(*===================================================================================================*)
(* Monitor reset conditions                                                                          *)
(*===================================================================================================*)
METHOD OkToReset : BOOL
VAR_INPUT
END_VAR
(*===================================================================================================*)
(* Monitor reset conditions                                                                          *)
(*===================================================================================================*)

OkToReset := ((StateAct = NLG_STATUS_STANDBY) AND   // Check for standby mode
			  (ResetCnt < 3));                      // Check reset count is less than 3
END_METHOD

END_FUNCTION_BLOCK

// Application/UserCode/MCU/MCU_Rx
PROGRAM MCU_Rx
VAR
	MCU_CommandResponse1_Rx		:	Receive_CAN1_STD;
	MCU_CommandResponse2_Rx		:	Receive_CAN1_STD;
	MCU_EventInfo1_Rx			:	Receive_CAN1_STD;
	MCU_Info1_Rx				:	Receive_CAN1_STD;
	MCU_Info2_Rx				:	Receive_CAN1_STD;
	MCU_OnEventInfo1_Rx			:	Receive_CAN1_STD;
	MCU_Thermal1_Rx				:	Receive_CAN1_STD;
	MCU_PollingMCUResponse_Rx	:	Receive_CAN1_STD;
	MCU_PollingVMU_Rx			:	Receive_CAN1_STD;
	
	MCU_CommandResponse1_Rx_Timer	:	TON;
	MCU_CommandResponse2_Rx_Timer	:	TON;
	MCU_EventInfo1_Rx_Timer			:	TON;
	MCU_Info1_Rx_Timer				:	TON;
	MCU_Info2_Rx_Timer				:	TON;
	MCU_Thermal1_Rx_Timer			:	TON;
END_VAR


MCU_CommandResponse1_Rx(u32_COBID	:=	16#043,
						 q_NewData => ,
						 au8_Data => ,
						 u8_Length => 			);
						 
MCU_CommandResponse2_Rx(u32_COBID	:=	16#044,
						 q_NewData => ,
						 au8_Data => ,
						 u8_Length => 			);
						 
MCU_EventInfo1_Rx(u32_COBID	:=	16#442,
						 q_NewData => ,
						 au8_Data => ,
						 u8_Length => 			);
						 
MCU_Info1_Rx(u32_COBID	:=	16#440,
						 q_NewData => ,
						 au8_Data => ,
						 u8_Length => 			);
						 
MCU_Info2_Rx(u32_COBID	:=	16#441,
						 q_NewData => ,
						 au8_Data => ,
						 u8_Length => 			);
						 
MCU_OnEventInfo1_Rx(u32_COBID	:=	16#443,
						 q_NewData => ,
						 au8_Data => ,
						 u8_Length => 			);
						 
MCU_Thermal1_Rx(u32_COBID	:=	16#449,
						 q_NewData => ,
						 au8_Data => ,
						 u8_Length => 			);
						 
MCU_PollingMCUResponse_Rx(u32_COBID	:=	16#448,
						 q_NewData => ,
						 au8_Data => ,
						 u8_Length => 			);
						 
MCU_PollingVMU_Rx(u32_COBID	:=	16#445,
						 q_NewData => ,
						 au8_Data => ,
						 u8_Length => 			);
						 


(*MCUCommandResponse1*)
gu8_MCU_State								:=	MCU_CommandResponse1_Rx.au8_Data[0] AND 2#00001111;
gu8_MCU_OperationalMode						:=	MCU_CommandResponse1_Rx.au8_Data[0] AND 2#01110000;
gq_MCU_RegenDeratingStatus					:=	MCU_CommandResponse1_Rx.au8_Data[0].7;
gu8_MCU_RegenDerating						:=	MCU_CommandResponse1_Rx.au8_Data[1] AND 2#00001111;
gu8_MCU_TractionDerating					:=	MCU_CommandResponse1_Rx.au8_Data[1] AND 2#11110000;
gu16_MCU_MaxMotorSpeedForward_Rx			:=	USINT_TO_UINT(MCU_CommandResponse1_Rx.au8_Data[2]) +
												SHL(BOOL_TO_UINT(MCU_CommandResponse1_Rx.au8_Data[3].0), 8);
gu16_MCU_MaxMotorSpeedReverse_Rx			:=	USINT_TO_UINT(MCU_CommandResponse1_Rx.au8_Data[4]) +
												SHL(BOOL_TO_UINT(MCU_CommandResponse1_Rx.au8_Data[5].0), 8);
gq_MCU_MaxMotorSpeedForwardStatus			:=	MCU_CommandResponse1_Rx.au8_Data[5].1;
gq_MCU_MaxMotorSpeedReverseStatus			:=	MCU_CommandResponse1_Rx.au8_Data[5].2;
gq_MCU_TractionDeratingStatus				:=	MCU_CommandResponse1_Rx.au8_Data[5].3;
gu8_MCU_RollingCounter_Comm1				:=	MCU_CommandResponse1_Rx.au8_Data[5] AND 2#11110000;
(*MCUCommandResponse2*)
gu16_MCU_MotorSpeed_Rx						:=	USINT_TO_UINT(MCU_CommandResponse2_Rx.au8_Data[0]) +
												SHL(USINT_TO_UINT(MCU_CommandResponse2_Rx.au8_Data[1]), 8);
gu16_MCU_MotorAngle_Rx						:=	USINT_TO_UINT(MCU_CommandResponse2_Rx.au8_Data[2]) +
												SHL(USINT_TO_UINT(MCU_CommandResponse2_Rx.au8_Data[3]), 8);
gq_MVU_MotorAngleStatus						:=	MCU_CommandResponse2_Rx.au8_Data[4].0;
gq_MCU_MotorSpeedStatus						:=	MCU_CommandResponse2_Rx.au8_Data[4].1;
gq_MCU_SpeedReductionRequest				:=	MCU_CommandResponse2_Rx.au8_Data[4].2;
gq_MCU_EmergencyStop						:=	MCU_CommandResponse2_Rx.au8_Data[4].3;
gu8_MCU_RollingCounter_Comm2				:=	MCU_CommandResponse2_Rx.au8_Data[4] AND 2#11110000;
(*MCUEventInfo1*)
gq_MCU_Fault_PhaseToChassis					:=	MCU_EventInfo1_Rx.au8_Data[0].0;
gq_MCU_Fault_InterlockBatteryCable			:=	MCU_EventInfo1_Rx.au8_Data[0].1;
gq_MCU_Fault_InterlockMotorCable			:=	MCU_EventInfo1_Rx.au8_Data[0].2;
gq_MCU_Fault_DriveCoverWasOpened			:=	MCU_EventInfo1_Rx.au8_Data[0].3;
gq_MCU_Fault_PhaseToChassisStatus			:=	MCU_EventInfo1_Rx.au8_Data[0].4;
gq_MCU_Fault_InterlockBatteryCableStatus	:=	MCU_EventInfo1_Rx.au8_Data[0].5;
gq_MCU_Fault_InterlockMotorCableStatus		:=	MCU_EventInfo1_Rx.au8_Data[0].6;
gq_MCU_Fault_DriveCoverWasOpenedStatus		:=	MCU_EventInfo1_Rx.au8_Data[0].7;
(*MCUInfo1*)
gu8_MCU_AuxiliaryVoltage_Rx					:=	MCU_Info1_Rx.au8_Data[0];
gu16_MCU_HighPowerVoltage					:=	USINT_TO_UINT(MCU_Info1_Rx.au8_Data[1]) +
												SHL(USINT_TO_UINT(MCU_Info1_Rx.au8_Data[2] AND 2#00000111), 8);
gq_MCU_HighPowerCurrentStatus				:=	MCU_Info1_Rx.au8_Data[2].3;
gq_MCU_AuxiliaryVoltageStatus				:=	MCU_Info1_Rx.au8_Data[2].4;
gq_MCU_HighPowerVoltageStatus				:=	MCU_Info1_Rx.au8_Data[2].5;
gu16_MCU_HighPowerCurrent_Rx				:=	USINT_TO_UINT(MCU_Info1_Rx.au8_Data[3]) +
												SHL(USINT_TO_UINT(MCU_Info1_Rx.au8_Data[4]), 8);
gu8_MCU_RollingCounter_Info1				:=	MCU_Info1_Rx.au8_Data[5];
(*MCUInfo2*)
gu16_MCU_MotorTorqueEstimated_Rx			:=	USINT_TO_UINT(MCU_Info2_Rx.au8_Data[0]) +
												SHL(USINT_TO_UINT(MCU_Info2_Rx.au8_Data[1]), 8);
gu16_MCU_TractionTorqueAvailable_Rx			:=	USINT_TO_UINT(MCU_Info2_Rx.au8_Data[2]) +
												SHL(USINT_TO_UINT(MCU_Info2_Rx.au8_Data[3] AND 2#01111111), 8);
gu16_MCU_RegenTorqueAvailable_Rx			:=	USINT_TO_UINT(MCU_Info2_Rx.au8_Data[4]) +
												SHL(USINT_TO_UINT(MCU_Info2_Rx.au8_Data[5] AND 2#01111111), 8);
gq_MCU_MotorTorqueEstimatedStatus			:=	MCU_Info2_Rx.au8_Data[6].1;
gq_MCU_TractionTorqueAvailableStatus		:=	MCU_Info2_Rx.au8_Data[6].2;
gq_MCU_RegenTorqueAvailableStatus			:=	MCU_Info2_Rx.au8_Data[6].3;
gu8_MCU_RollingCounter_Info2				:=	MCU_Info2_Rx.au8_Data[6] AND 2#11110000;
(*MCUOnEventInfo1*)
gu16_MCU_EventID							:=	USINT_TO_UINT(MCU_OnEventInfo1_Rx.au8_Data[0]) +
												SHL(USINT_TO_UINT(MCU_OnEventInfo1_Rx.au8_Data[1]), 8);
gu8_MCU_RollingCounter_OnEventInfo1			:=	MCU_OnEventInfo1_Rx.au8_Data[4] AND 2#11110000;
(*MCUThermal1*)
gu8_MCU_DriveCoolingFlowRequest_Rx			:=	MCU_Thermal1_Rx.au8_Data[0];
gu8_MCU_MotorCoolingFlowRequest_Rx			:=	MCU_Thermal1_Rx.au8_Data[1];
gu8_MCU_ThermalIndicator_Rx					:=	MCU_Thermal1_Rx.au8_Data[2];
gq_MCU_DriveCoolingFlowRequestStatus		:=	MCU_Thermal1_Rx.au8_Data[3].0;
gq_MCU_MotorCoolingFlowRequestStatus		:=	MCU_Thermal1_Rx.au8_Data[3].1;
gq_MCU_ThermalIndicatorStatus				:=	MCU_Thermal1_Rx.au8_Data[3].2;
gu8_MCU_RollingCounter_Thermal1				:=	MCU_Thermal1_Rx.au8_Data[3] AND 2#11110000;
(*MCUPollingMCUResponse*)
gq_MCU_ResponseAcknowledgement				:=	MCU_PollingMCUResponse_Rx.au8_Data[0].0;
gu8_MCU_MCUPollResponse_Multiplex			:=	MCU_PollingMCUResponse_Rx.au8_Data[0] AND 2#01111111;
CASE gu8_MCU_MCUPollResponse_Multiplex OF
	MAXMOTORSPEED:	(*MCU MaxMotorSpeed*)
		gu16_MCU_MaxMotorSpeed_Rx			:=	USINT_TO_UINT(MCU_PollingMCUResponse_Rx.au8_Data[1]) +
												SHL(USINT_TO_UINT(MCU_PollingMCUResponse_Rx.au8_Data[2]), 8);
	MAXMOTORTORQUE:	(*MCU MaxMotorTorque*)
		gu16_MCU_MaxMotorTorque_Rx			:=	USINT_TO_UINT(MCU_PollingMCUResponse_Rx.au8_Data[1]) +
												SHL(USINT_TO_UINT(MCU_PollingMCUResponse_Rx.au8_Data[2] AND 2#01111111), 8);
	PROTOCOLVERSION:	(*MCU ProtocolVersion*)
		gu8_MCU_MajorMCUProtocol			:=	MCU_PollingMCUResponse_Rx.au8_Data[1];
		gu8_MCU_MinorMCUProtocol			:=	MCU_PollingMCUResponse_Rx.au8_Data[2];
		gu8_MCU_ExtensionMajor				:=	MCU_PollingMCUResponse_Rx.au8_Data[3];
		gu8_MCU_ExtensionMinor				:=	MCU_PollingMCUResponse_Rx.au8_Data[4];
	SWVERSION1:	(*MCU SWVersion1*)
		gu8_MCU_MajorMCUSW					:=	MCU_PollingMCUResponse_Rx.au8_Data[1];
		gu8_MCU_MinorMCUSW					:=	MCU_PollingMCUResponse_Rx.au8_Data[2];
		gu16_MCU_BranchMCUSW				:=	USINT_TO_UINT(MCU_PollingMCUResponse_Rx.au8_Data[3]) +
												SHL(USINT_TO_UINT(MCU_PollingMCUResponse_Rx.au8_Data[4]), 8);
	SWVERSION2	:(*MCU SWVersion2*)
		gu32_MCU_RevisionMCUSW				:=	USINT_TO_UDINT(MCU_PollingMCUResponse_Rx.au8_Data[1]) +
												SHL(USINT_TO_UDINT(MCU_PollingMCUResponse_Rx.au8_Data[2]), 8) +
												SHL(USINT_TO_UDINT(MCU_PollingMCUResponse_Rx.au8_Data[3]), 16) +
												SHL(USINT_TO_UDINT(MCU_PollingMCUResponse_Rx.au8_Data[4]), 24);
	TOTALMOTORROTATION:	(*MCU TotalMotorRotation*)
		gu32_MCU_TotalMotorRotation_LSB			:=	USINT_TO_UDINT(MCU_PollingMCUResponse_Rx.au8_Data[1]) +
												SHL(USINT_TO_UDINT(MCU_PollingMCUResponse_Rx.au8_Data[2]), 8) +
												SHL(USINT_TO_UDINT(MCU_PollingMCUResponse_Rx.au8_Data[3]), 16) +
												SHL(USINT_TO_UDINT(MCU_PollingMCUResponse_Rx.au8_Data[4]), 24);
		gu32_MCU_TotalMotorRotation_MSB			:=	USINT_TO_UDINT(MCU_PollingMCUResponse_Rx.au8_Data[5]) +
												SHL(USINT_TO_UDINT(MCU_PollingMCUResponse_Rx.au8_Data[6]), 8);
	TOTALMOTORROTATIONUSINTMCU:	(*MCU TotalMotorRotationUsingMCU*)
	;
ELSE
	;
END_CASE
	
(*MCUPollingVMU*)
gu8_MCU_VMUBootNumber						:=	MCU_PollingVMU_Rx.au8_Data[0];
CASE gu8_MCU_VMUBootNumber OF
	VMUBOOTNUMBER:	(*VMUBootNumber*)
		gu16_MCU_BootNumber						:=	USINT_TO_UINT(MCU_PollingVMU_Rx.au8_Data[1]) +
													SHL(USINT_TO_UINT(MCU_PollingVMU_Rx.au8_Data[2]), 8);
ELSE
	;
END_CASE
	
MCU_CommandResponse1_Rx_Timer(IN := NOT(MCU_CommandResponse1_Rx.q_NewData), PT := T#3S);
MCU_CommandResponse2_Rx_Timer(IN := NOT(MCU_CommandResponse2_Rx.q_NewData), PT := T#3S);
MCU_EventInfo1_Rx_Timer(IN := NOT(MCU_EventInfo1_Rx.q_NewData), PT := T#3S);
MCU_Info1_Rx_Timer(IN := NOT(MCU_Info1_Rx.q_NewData), PT := T#3S);
MCU_Info2_Rx_Timer(IN := NOT(MCU_Info2_Rx.q_NewData), PT := T#3S);
MCU_Thermal1_Rx_Timer(IN := NOT(MCU_Thermal1_Rx.q_NewData), PT := T#3S);
IF (MCU_CommandResponse1_Rx_Timer.Q = TRUE AND MCU_CommandResponse2_Rx_Timer.Q = TRUE AND MCU_EventInfo1_Rx_Timer.Q = TRUE AND
	MCU_Info1_Rx_Timer.Q = TRUE AND MCU_Info2_Rx_Timer.Q = TRUE AND MCU_Thermal1_Rx_Timer.Q = TRUE) THEN
	gq_MCU_CommsLoss	:=	TRUE;
ELSE
	gq_MCU_CommsLoss	:=	FALSE;
END_IF



MCU_RxConversion();

END_PROGRAM

// Application/UserCode/MCU/MCU_RxConversion
PROGRAM MCU_RxConversion
VAR
END_VAR
VAR CONSTANT
	MAXSPEED_CF		:	USINT	:=	100;
	UINT_OFFSET_CF	:	UINT	:=	32767;
	QUARTER_CF		:	REAL	:=	0.25;
	EIGHTH_CF		:	REAL	:=	0.125;
	UINT_MAX		:	UDINT	:=	65536;
	MCU_CF			:	REAL	:=	0.78125;
	CF_2POW11		:	UINT	:=	2048;
	CF_2POW12		:	UINT	:=	4096;
	
	MAX_UDINT		:	REAL	:=	4294967296;
END_VAR



gr_MCU_MaxMotorSpeedForward		:=	UINT_TO_REAL(gu16_MCU_MaxMotorSpeedForward_Rx) * MAXSPEED_CF;
gr_MCU_MaxMotorSpeedReverse		:=	UINT_TO_REAL(gu16_MCU_MaxMotorSpeedReverse_Rx) * MAXSPEED_CF;
gr_MCU_MotorSpeed				:=	UINT_TO_REAL(gu16_MCU_MotorSpeed_Rx) - UINT_OFFSET_CF;
gr_MCU_MotorAngle				:=	UINT_TO_REAL(gu16_MCU_MotorAngle_Rx) / UDINT_TO_REAL(UINT_MAX);
gr_MCU_AuxiliaryVoltage			:=	USINT_TO_REAL(gu8_MCU_AuxiliaryVoltage_Rx) * QUARTER_CF;
gr_MCU_HighPowerCurrent			:=	UINT_TO_REAL(gu16_MCU_HighPowerCurrent_Rx) * QUARTER_CF - CF_2POW11;
gr_MCU_MotorTorqueEstimated		:=	UINT_TO_REAL(gu16_MCU_MotorTorqueEstimated_Rx) * EIGHTH_CF - CF_2POW12;
gr_MCU_TractionTorqueAvailable	:=	UINT_TO_REAL(gu16_MCU_TractionTorqueAvailable_Rx) * EIGHTH_CF;
gr_MCU_RegenTorqueAvailable		:=	UINT_TO_REAL(gu16_MCU_RegenTorqueAvailable_Rx) * EIGHTH_CF;
gr_MCU_DriveCoolingFlowRequest	:=	USINT_TO_REAL(gu8_MCU_DriveCoolingFlowRequest_Rx) * MCU_CF;
gr_MCU_MotorCoolingFlowRequest	:=	USINT_TO_REAL(gu8_MCU_MotorCoolingFlowRequest_Rx) * MCU_CF;
gr_MCU_ThermalIndicator			:=	USINT_TO_REAL(gu8_MCU_ThermalIndicator_Rx) * MCU_CF;
gr_MCU_MaxMotorSpeed			:=	UINT_TO_REAL(gu16_MCU_MaxMotorSpeed_Rx) - UINT_OFFSET_CF;
gr_MCU_MaxMotorTorque			:=	UINT_TO_REAL(gu16_MCU_MaxMotorTorque_Rx) * EIGHTH_CF;

gr_MCU_TotalMotorRotation_LSB	:=	UDINT_TO_REAL(gu32_MCU_TotalMotorRotation_LSB);
gr_MCU_TotalMotorRotation_MSB	:=	UDINT_TO_REAL(gu32_MCU_TotalMotorRotation_MSB) * MAX_UDINT;
gr_MCU_TotalMotorRotation		:=	gr_MCU_TotalMotorRotation_LSB + gr_MCU_TotalMotorRotation_MSB;

END_PROGRAM

// Application/UserCode/CAN Function Blocks/CAN1/Receive_CAN1_STD
FUNCTION_BLOCK Receive_CAN1_STD
VAR_INPUT
	u32_COBID	:	DWORD;
END_VAR
VAR_OUTPUT
	q_NewData	:	BOOL;
	au8_Data	:	ARRAY [0..7] OF BYTE;
	u8_Length	:	BYTE;
END_VAR
VAR
	hq_Initialise	:	BOOL	:=	FALSE;
	ht_RxMessage	:	t_CANReceive;
	ht_MsgRx		:	Callback_Receive_CAN1;
END_VAR



IF (hq_Initialise = FALSE) THEN
	
	(*11 bit*)
	G_CAN1_Channel.AddCOBID(i_CobId := u32_COBID,
							i_itfCallback := ht_MsgRx,
							i_Argument := ADR(ht_RxMessage));
	(*
	(*29 bit*)
	G_CAN1_Channel.AddCOBID(i_CobId := u32_COBID OR EPEC_CANVXD.MASK_29BIT,
							i_itfCallback := ht_MsgRx,
							i_Argument := ADR(ht_RxMessage));
*)	(*G_CAN1_Channel.SetMask(i_CobID := u32_COBID OR EPEC_CANVXD.MASK_29BIT, i_Mask := 16#0C009000 OR EPEC_CANVXD.MASK_29BIT);
*)
	hq_Initialise	:=	TRUE;
END_IF


IF (ht_RxMessage.q_NewDataRxed = TRUE) THEN
	au8_Data	:=	ht_RxMessage.Data;
	u8_Length	:=	ht_RxMessage.Len;
	q_NewData	:=	TRUE;
	ht_RxMessage.q_NewDataRxed	:=	FALSE;
ELSE
	q_NewData	:=	FALSE;
END_IF

END_FUNCTION_BLOCK

// Application/UserCode/BMS/OrionBMS/OrionBMS1_Rx
PROGRAM OrionBMS1_Rx
VAR
	OrionBMS1_6B0_Rx	:	Receive_CAN2_STD;
	OrionBMS1_6B1_Rx	:	Receive_CAN2_STD;
	OrionBMS1_6B2_Rx	:	Receive_CAN2_STD;
	OrionBMS1_6B3_Rx	:	Receive_CAN2_STD;
	OrionBMS1_6B4_Rx	:	Receive_CAN2_STD;
	OrionBMS1_6B5_Rx	:	Receive_CAN2_STD;
	OrionBMS1_6B6_Rx	:	Receive_CAN2_STD;
	OrionBMS1_6B7_Rx	:	Receive_CAN2_STD;
	OrionBMS1_6B8_Rx	:	Receive_CAN2_STD;
	OrionBMS1_6B9_Rx	:	Receive_CAN2_STD;
	OrionBMS1_6BA_Rx	:	Receive_CAN2_STD;
	OrionBMS1_6BB_Rx	:	Receive_CAN2_STD;
	OrionBMS1_6BC_Rx	:	Receive_CAN2_STD;
	OrionBMS1_6BD_Rx	:	Receive_CAN2_STD;
	
	OrionBMS1_6B0_Rx_Timer	:	TON;
	OrionBMS1_6B1_Rx_Timer	:	TON;
	OrionBMS1_6B2_Rx_Timer	:	TON;
	OrionBMS1_6B3_Rx_Timer	:	TON;
	OrionBMS1_6B4_Rx_Timer	:	TON;
	OrionBMS1_6B5_Rx_Timer	:	TON;
	OrionBMS1_6B6_Rx_Timer	:	TON;
	OrionBMS1_6B7_Rx_Timer	:	TON;
	OrionBMS1_6B8_Rx_Timer	:	TON;
	OrionBMS1_6B9_Rx_Timer	:	TON;
	OrionBMS1_6BA_Rx_Timer	:	TON;
	OrionBMS1_6BB_Rx_Timer	:	TON;
	OrionBMS1_6BC_Rx_Timer	:	TON;
	OrionBMS1_6BD_Rx_Timer	:	TON;
	END_VAR

(*Program to receive all data from the Orion BMS*)
(*Initial saving CAN messages to receipt strucutres*)
OrionBMS1_6B0_Rx(u32_COBID	:=	16#6B0,
				 q_NewData => ,
				 au8_Data => ,
				 u8_Length => 			);
				 
OrionBMS1_6B1_Rx(u32_COBID	:=	16#6B1,
				 q_NewData => ,
				 au8_Data => ,
				 u8_Length => 			);
				 
OrionBMS1_6B2_Rx(u32_COBID	:=	16#6B2,
				 q_NewData => ,
				 au8_Data => ,
				 u8_Length => 			);
				 
OrionBMS1_6B3_Rx(u32_COBID	:=	16#6B3,
				 q_NewData => ,
				 au8_Data => ,
				 u8_Length => 			);
				 
OrionBMS1_6B4_Rx(u32_COBID	:=	16#6B4,
				 q_NewData => ,
				 au8_Data => ,
				 u8_Length => 			);
				 
OrionBMS1_6B5_Rx(u32_COBID	:=	16#6B5,
				 q_NewData => ,
				 au8_Data => ,
				 u8_Length => 			);
				 
OrionBMS1_6B6_Rx(u32_COBID	:=	16#6B6,
				 q_NewData => ,
				 au8_Data => ,
				 u8_Length => 			);
				 
OrionBMS1_6B7_Rx(u32_COBID	:=	16#6B7,
				 q_NewData => ,
				 au8_Data => ,
				 u8_Length => 			);
			 
OrionBMS1_6B8_Rx(u32_COBID	:=	16#6B8,
				 q_NewData => ,
				 au8_Data => ,
				 u8_Length => 			);
				 
OrionBMS1_6B9_Rx(u32_COBID	:=	16#6B9,
				 q_NewData => ,
				 au8_Data => ,
				 u8_Length => 			);
				 
OrionBMS1_6BA_Rx(u32_COBID	:=	16#6BA,
				 q_NewData => ,
				 au8_Data => ,
				 u8_Length => 			);
				 
OrionBMS1_6BB_Rx(u32_COBID	:=	16#6BB,
				 q_NewData => ,
				 au8_Data => ,
				 u8_Length => 			);
				 
OrionBMS1_6BC_Rx(u32_COBID	:=	16#6BC,
				 q_NewData => ,
				 au8_Data => ,
				 u8_Length => 			);
				 
OrionBMS1_6BD_Rx(u32_COBID	:=	16#6BD,
				 q_NewData => ,
				 au8_Data => ,
				 u8_Length => 			);


(*Unpacking structures into variables*)
(*6B0*)
gs16_OrionBMS1_PackCurrent	:=	USINT_TO_INT(OrionBMS1_6B0_Rx.au8_Data[0]) +
								SHL(USINT_TO_INT(OrionBMS1_6B0_Rx.au8_Data[1]), 8);
gu16_OrionBMS1_RAW_Pack_Voltage	:=	USINT_TO_UINT(OrionBMS1_6B0_Rx.au8_Data[2]) +
								SHL(USINT_TO_UINT(OrionBMS1_6B0_Rx.au8_Data[3]), 8);
gu8_OrionBMS1_RAW_SOC	:=	OrionBMS1_6B0_Rx.au8_Data[4];
gu16_OrionBMS1_RelayState	:=	USINT_TO_UINT(OrionBMS1_6B0_Rx.au8_Data[5]) +
								SHL(USINT_TO_UINT(OrionBMS1_6B0_Rx.au8_Data[6]), 8);
gu8_OrionBMS1_Custom_Flag_1	:=	OrionBMS1_6B0_Rx.au8_Data[7];

(*6B1*)
gu8_OrionBMS1_Isolation_ADC			:=	USINT_TO_UINT(OrionBMS1_6B1_Rx.au8_Data[0]) +
									SHL(USINT_TO_UINT(OrionBMS1_6B1_Rx.au8_Data[1]), 8);
gu8_OrionBMS1_Shortest_Wave			:=	USINT_TO_UINT(OrionBMS1_6B1_Rx.au8_Data[2]) +
									SHL(USINT_TO_UINT(OrionBMS1_6B1_Rx.au8_Data[3]), 8);
gu16_OrionBMS1_Isolation_Clipping	:=	USINT_TO_UINT(OrionBMS1_6B1_Rx.au8_Data[4]) +
									SHL(USINT_TO_UINT(OrionBMS1_6B1_Rx.au8_Data[5]), 8);
gu16_OrionBMS1_Isolation_Threshold	:=	USINT_TO_UINT(OrionBMS1_6B1_Rx.au8_Data[6]) +
									SHL(USINT_TO_UINT(OrionBMS1_6B1_Rx.au8_Data[7]), 8);
									
(*6B2*)
gu16_OrionBMS1_DTC_Flags1		:=	USINT_TO_UINT(OrionBMS1_6B2_Rx.au8_Data[0]) +
								SHL(USINT_TO_UINT(OrionBMS1_6B2_Rx.au8_Data[1]), 8);
gu16_OrionBMS1_DTC_Flags2		:=	USINT_TO_UINT(OrionBMS1_6B2_Rx.au8_Data[2]) +
								SHL(USINT_TO_UINT(OrionBMS1_6B2_Rx.au8_Data[3]), 8);
gu16_OrionBMS1_FailsafeStatus	:=	USINT_TO_UINT(OrionBMS1_6B2_Rx.au8_Data[4]) +
								SHL(USINT_TO_UINT(OrionBMS1_6B2_Rx.au8_Data[5]), 8);
gu16_OrionBMS1_Current_Limit_Status		:=	USINT_TO_UINT(OrionBMS1_6B2_Rx.au8_Data[6]) +
								SHL(USINT_TO_UINT(OrionBMS1_6B2_Rx.au8_Data[7]), 8);
(*6B3*)
gu8_OrionBMS1_PackHealth			:=	OrionBMS1_6B3_Rx.au8_Data[0];
gu16_OrionBMS1_PackCycles			:=	USINT_TO_UINT(OrionBMS1_6B3_Rx.au8_Data[1]) +
									SHL(USINT_TO_UINT(OrionBMS1_6B3_Rx.au8_Data[2]), 8);
gu16_OrionBMS1_PackResistance		:=	USINT_TO_UINT(OrionBMS1_6B3_Rx.au8_Data[3]) +
									SHL(USINT_TO_UINT(OrionBMS1_6B3_Rx.au8_Data[4]), 8);
gu8_OrionBMS1_PopulatedCells		:=	OrionBMS1_6B3_Rx.au8_Data[5];
gu16_OrionBMS1_MaximumPackVoltage	:=	USINT_TO_UINT (OrionBMS1_6B3_Rx.au8_Data[6]) +
									SHL(USINT_TO_UINT(OrionBMS1_6B3_Rx.au8_Data[7]),8);

(*6B4*)
gu8_OrionBMS1_HighTemp		:=	OrionBMS1_6B4_Rx.au8_Data[0];
gu8_OrionBMS1_LowTemp		:=	OrionBMS1_6B4_Rx.au8_Data[1];
gu8_OrionBMS1_AverageTemp	:=	OrionBMS1_6B4_Rx.au8_Data[2];
gu8_OrionBMS1_InternalTemp	:=	OrionBMS1_6B4_Rx.au8_Data[3];
gu16_OrionBMS1_MinimumPackVoltage	:=	USINT_TO_UINT(OrionBMS1_6B4_Rx.au8_Data[4]) +
									SHL(USINT_TO_UINT(OrionBMS1_6B4_Rx.au8_Data[5]), 8);
gu16_OrionBMS1_PackAmphours	:=	USINT_TO_UINT(OrionBMS1_6B4_Rx.au8_Data[6]) +
								SHL(USINT_TO_UINT(OrionBMS1_6B4_Rx.au8_Data[7]), 8);
(*6B5*)
gu16_OrionBMS1_AverageCellVoltage	:=	USINT_TO_UINT(OrionBMS1_6B5_Rx.au8_Data[0]) +
										SHL(USINT_TO_UINT(OrionBMS1_6B5_Rx.au8_Data[1]), 8);
gu16_OrionBMS1_LowCellVoltage		:=	USINT_TO_UINT(OrionBMS1_6B5_Rx.au8_Data[2]) +
										SHL(USINT_TO_UINT(OrionBMS1_6B5_Rx.au8_Data[3]), 8);
gu16_OrionBMS1_HighCellVoltage		:=	USINT_TO_UINT(OrionBMS1_6B5_Rx.au8_Data[4]) +
										SHL(USINT_TO_UINT(OrionBMS1_6B5_Rx.au8_Data[5]), 8);
gu8_OrionBMS1_LowCellVoltNumber		:=	OrionBMS1_6B5_Rx.au8_Data[6];
gu8_OrionBMS1_HighCellVoltNumber	:=	OrionBMS1_6B5_Rx.au8_Data[7];
(*6B6*)
gu8_OrionBMS1_Low_Intres_ID			:=	OrionBMS1_6B6_Rx.au8_Data[0];
gu8_OrionBMS1_High_Intres_ID		:=	OrionBMS1_6B6_Rx.au8_Data[1];
gu16_OrionBMS1_Low_Cell_Resistance	:=	USINT_TO_UINT(OrionBMS1_6B6_Rx.au8_Data[2]) +
										SHL(USINT_TO_UINT(OrionBMS1_6B6_Rx.au8_Data[3]), 8);
gu16_OrionBMS1_High_Cell_Resistance	:=	USINT_TO_UINT(OrionBMS1_6B6_Rx.au8_Data[4]) +
										SHL(USINT_TO_UINT(OrionBMS1_6B6_Rx.au8_Data[5]), 8);
gu16_OrionBMS1_Average_Cell_Resistance	:=	USINT_TO_UINT(OrionBMS1_6B6_Rx.au8_Data[6]) +
										SHL(USINT_TO_UINT(OrionBMS1_6B6_Rx.au8_Data[7]), 8);

(*6B7*)
gu8_OrionBMS1_Low_Thermistor_ID			:=	OrionBMS1_6B7_Rx.au8_Data[0];
gu8_OrionBMS1_High_Thermistor_ID		:=	OrionBMS1_6B7_Rx.au8_Data[1];
gu16_OrionBMS1_PackDCL				:=	USINT_TO_UINT(OrionBMS1_6B7_Rx.au8_Data[2]) +
										SHL(USINT_TO_UINT(OrionBMS1_6B7_Rx.au8_Data[3]), 8);
gu16_OrionBMS1_PackCCL				:=	USINT_TO_UINT(OrionBMS1_6B7_Rx.au8_Data[4]) +
										SHL(USINT_TO_UINT(OrionBMS1_6B7_Rx.au8_Data[5]), 8);
gu16_OrionBMS1_PackSummedVoltage	:=	USINT_TO_UINT(OrionBMS1_6B7_Rx.au8_Data[6]) +
										SHL(USINT_TO_UINT(OrionBMS1_6B7_Rx.au8_Data[7]), 8);

(*6B8*)
	gu8_OrionBMS1_Firmware_Minor		:=	OrionBMS1_6B8_Rx.au8_Data[0];	
	gu8_OrionBMS1_Firmware_Patch		:=	OrionBMS1_6B8_Rx.au8_Data[1];		
	gu8_OrionBMS1_Constant_2			:=	OrionBMS1_6B8_Rx.au8_Data[2];		
	gu8_OrionBMS1_Constant_3			:=	OrionBMS1_6B8_Rx.au8_Data[3];		
	gu8_OrionBMS1_Constant_4			:=	OrionBMS1_6B8_Rx.au8_Data[4];		
	gu16_OrionBMS1_CheckSum	:=	USINT_TO_UINT(OrionBMS1_6B8_Rx.au8_Data[5]) +
										SHL(USINT_TO_UINT(OrionBMS1_6B8_Rx.au8_Data[6]), 8);
	gu8_OrionBMS1_Spare_6B6_7			:=	OrionBMS1_6B8_Rx.au8_Data[7];


(*6B9*)
gu8_OrionBMS1_6B9_0		:=	OrionBMS1_6B9_Rx.au8_Data[0];
gu8_OrionBMS1_6B9_1		:=	OrionBMS1_6B9_Rx.au8_Data[1];
gu8_OrionBMS1_6B9_2		:=	OrionBMS1_6B9_Rx.au8_Data[2];
gu8_OrionBMS1_6B9_3		:=	OrionBMS1_6B9_Rx.au8_Data[3];
gu8_OrionBMS1_6B9_4		:=	OrionBMS1_6B9_Rx.au8_Data[4];
gu8_OrionBMS1_6B9_5		:=	OrionBMS1_6B9_Rx.au8_Data[5];
gu8_OrionBMS1_6B9_6		:=	OrionBMS1_6B9_Rx.au8_Data[6];
gu8_OrionBMS1_6B9_7		:=	OrionBMS1_6B9_Rx.au8_Data[7];


(*6BA*)
gu8_OrionBMS1_6BA_0		:=	OrionBMS1_6BA_Rx.au8_Data[0];
gu8_OrionBMS1_6BA_1		:=	OrionBMS1_6BA_Rx.au8_Data[1];
gu8_OrionBMS1_6BA_2		:=	OrionBMS1_6BA_Rx.au8_Data[2];
gu8_OrionBMS1_6BA_3		:=	OrionBMS1_6BA_Rx.au8_Data[3];
gu8_OrionBMS1_6BA_4		:=	OrionBMS1_6BA_Rx.au8_Data[4];
gu8_OrionBMS1_6BA_5		:=	OrionBMS1_6BA_Rx.au8_Data[5];
gu8_OrionBMS1_6BA_6		:=	OrionBMS1_6BA_Rx.au8_Data[6];
gu8_OrionBMS1_6BA_7		:=	OrionBMS1_6BA_Rx.au8_Data[7];

(*6BB*)
gu8_OrionBMS1_6BB_0		:=	OrionBMS1_6BB_Rx.au8_Data[0];
gu8_OrionBMS1_6BB_1		:=	OrionBMS1_6BB_Rx.au8_Data[1];
gu8_OrionBMS1_6BB_2		:=	OrionBMS1_6BB_Rx.au8_Data[2];
gu8_OrionBMS1_6BB_3		:=	OrionBMS1_6BB_Rx.au8_Data[3];
gu8_OrionBMS1_6BB_4		:=	OrionBMS1_6BB_Rx.au8_Data[4];
gu8_OrionBMS1_6BB_5		:=	OrionBMS1_6BB_Rx.au8_Data[5];
gu8_OrionBMS1_6BB_6		:=	OrionBMS1_6BB_Rx.au8_Data[6];
gu8_OrionBMS1_6BB_7		:=	OrionBMS1_6BB_Rx.au8_Data[7];

(*6BC*)
gu8_OrionBMS1_6BC_0		:=	OrionBMS1_6BC_Rx.au8_Data[0];
gu8_OrionBMS1_6BC_1		:=	OrionBMS1_6BC_Rx.au8_Data[1];
gu8_OrionBMS1_6BC_2		:=	OrionBMS1_6BC_Rx.au8_Data[2];
gu8_OrionBMS1_6BC_3		:=	OrionBMS1_6BC_Rx.au8_Data[3];
gu8_OrionBMS1_6BC_4		:=	OrionBMS1_6BC_Rx.au8_Data[4];
gu8_OrionBMS1_6BC_5		:=	OrionBMS1_6BC_Rx.au8_Data[5];
gu8_OrionBMS1_6BC_6		:=	OrionBMS1_6BC_Rx.au8_Data[6];
gu8_OrionBMS1_6BC_7		:=	OrionBMS1_6BC_Rx.au8_Data[7];	
	
(*6BD*)
gu8_OrionBMS1_6BD_0		:=	OrionBMS1_6BD_Rx.au8_Data[0];
gu8_OrionBMS1_6BD_1		:=	OrionBMS1_6BD_Rx.au8_Data[1];
gu8_OrionBMS1_6BD_2		:=	OrionBMS1_6BD_Rx.au8_Data[2];
gu8_OrionBMS1_6BD_3		:=	OrionBMS1_6BD_Rx.au8_Data[3];
gu8_OrionBMS1_6BD_4		:=	OrionBMS1_6BD_Rx.au8_Data[4];
gu8_OrionBMS1_6BD_5		:=	OrionBMS1_6BD_Rx.au8_Data[5];
gu8_OrionBMS1_6BD_6		:=	OrionBMS1_6BD_Rx.au8_Data[6];
gu8_OrionBMS1_6BD_7		:=	OrionBMS1_6BD_Rx.au8_Data[7];

(*Comms loss check to ensure all messages are still being received*)
OrionBMS1_6B0_Rx_Timer(IN := NOT(OrionBMS1_6B0_Rx.q_NewData), PT := T#3S);
OrionBMS1_6B1_Rx_Timer(IN := NOT(OrionBMS1_6B1_Rx.q_NewData), PT := T#3S);
OrionBMS1_6B2_Rx_Timer(IN := NOT(OrionBMS1_6B2_Rx.q_NewData), PT := T#3S);
OrionBMS1_6B3_Rx_Timer(IN := NOT(OrionBMS1_6B3_Rx.q_NewData), PT := T#3S);
OrionBMS1_6B4_Rx_Timer(IN := NOT(OrionBMS1_6B4_Rx.q_NewData), PT := T#3S);
OrionBMS1_6B5_Rx_Timer(IN := NOT(OrionBMS1_6B5_Rx.q_NewData), PT := T#3S);
OrionBMS1_6B6_Rx_Timer(IN := NOT(OrionBMS1_6B6_Rx.q_NewData), PT := T#3S);
OrionBMS1_6B7_Rx_Timer(IN := NOT(OrionBMS1_6B7_Rx.q_NewData), PT := T#3S);
OrionBMS1_6B8_Rx_Timer(IN := NOT(OrionBMS1_6B8_Rx.q_NewData), PT := T#3S);
OrionBMS1_6B9_Rx_Timer(IN := NOT(OrionBMS1_6B9_Rx.q_NewData), PT := T#3S);
OrionBMS1_6BA_Rx_Timer(IN := NOT(OrionBMS1_6BA_Rx.q_NewData), PT := T#3S);
OrionBMS1_6BB_Rx_Timer(IN := NOT(OrionBMS1_6BB_Rx.q_NewData), PT := T#3S);
OrionBMS1_6BC_Rx_Timer(IN := NOT(OrionBMS1_6BC_Rx.q_NewData), PT := T#3S);
OrionBMS1_6BD_Rx_Timer(IN := NOT(OrionBMS1_6BD_Rx.q_NewData), PT := T#3S);
IF (OrionBMS1_6B0_Rx_Timer.Q = TRUE AND OrionBMS1_6B1_Rx_Timer.Q = TRUE AND OrionBMS1_6B2_Rx_Timer.Q = TRUE AND
	OrionBMS1_6B3_Rx_Timer.Q = TRUE AND OrionBMS1_6B4_Rx_Timer.Q = TRUE AND OrionBMS1_6B5_Rx_Timer.Q = TRUE AND
	OrionBMS1_6B6_Rx_Timer.Q = TRUE AND OrionBMS1_6B7_Rx_Timer.Q = TRUE AND OrionBMS1_6B8_Rx_Timer.Q = TRUE AND
	OrionBMS1_6B9_Rx_Timer.Q = TRUE AND OrionBMS1_6BA_Rx_Timer.Q = TRUE AND OrionBMS1_6BB_Rx_Timer.Q = TRUE AND
	OrionBMS1_6BC_Rx_Timer.Q = TRUE AND OrionBMS1_6BD_Rx_Timer.Q = TRUE											) THEN

	gq_OrionBMS1_CommsLoss	:=	TRUE;
ELSE
	gq_OrionBMS1_CommsLoss	:=	FALSE;
END_IF


OrionBMS1_RxConversion();

END_PROGRAM

// Application/UserCode/BMS/OrionBMS/OrionBMS1_RxConversion
PROGRAM OrionBMS1_RxConversion
VAR
	Safety_OK   : BOOL;
END_VAR
VAR CONSTANT
	SYSTEMRX_CF	:	REAL	:=	0.1;
	CURRENT_CF	:	REAL	:=	0.1;
END_VAR

(*Convert input variables into real units by applying conversion factors and offsets*)

gr_OrionBMS1_PackVoltage			:=	UINT_TO_REAL(gu16_OrionBMS1_RAW_Pack_Voltage) * SYSTEMRX_CF;
gr_OrionBMS1_PackCurrent			:=	INT_TO_REAL(gs16_OrionBMS1_PackCurrent) * CURRENT_CF;
gr_OrionBMS1_PackSOC				:=	REAL_TO_USINT(gu8_OrionBMS1_RAW_SOC / 2);
gr_OrionBMS1_Max_Charging_Voltage	:= gu8_OrionBMS1_PopulatedCells *3.65;

OrionBMS1_DTCFlag1_0A07_DischargeLimitEnforcementFault1		:=	gu16_OrionBMS1_DTC_Flags1.0;
OrionBMS1_DTCFlag1_0A08_ChargerSafetyRelayFault1 			:=	gu16_OrionBMS1_DTC_Flags1.1;
OrionBMS1_DTCFlag1_0A09_InternalHardwareFault1				:=	gu16_OrionBMS1_DTC_Flags1.2;
OrionBMS1_DTCFlag1_0A0A_InternalHeatskinkThermistorFault 	:=	gu16_OrionBMS1_DTC_Flags1.3;
OrionBMS1_DTCFlag1_0A0B_InternalSoftwareFault1				:=	gu16_OrionBMS1_DTC_Flags1.4;
OrionBMS1_DTCFlag1_0A0C_HighestCellVoltageTooHighFault1 	:=	gu16_OrionBMS1_DTC_Flags1.5;
OrionBMS1_DTCFlag1_0A0E_LowestCellVoltageTooLowFault 		:=	gu16_OrionBMS1_DTC_Flags1.6;
OrionBMS1_DTCFlag1_0A10_PackTooHotFault1 					:=	gu16_OrionBMS1_DTC_Flags1.7;
OrionBMS1_DTCFlags_Reserved_Bit8 							:=	gu16_OrionBMS1_DTC_Flags1.8;
OrionBMS1_DTCFlags_Reserved_Bit9 							:=	gu16_OrionBMS1_DTC_Flags1.9;
OrionBMS1_DTCFlags_Reserved_Bit10 							:=	gu16_OrionBMS1_DTC_Flags1.10;
OrionBMS1_DTCFlags_Reserved_Bit11 							:=	gu16_OrionBMS1_DTC_Flags1.11;
OrionBMS1_DTCFlags_Reserved_Bit12 							:=	gu16_OrionBMS1_DTC_Flags1.12;
OrionBMS1_DTCFlags_Reserved_Bit13 							:=	gu16_OrionBMS1_DTC_Flags1.13;
OrionBMS1_DTCFlags_Reserved_Bit14 							:=	gu16_OrionBMS1_DTC_Flags1.14;
OrionBMS1_DTCFlags_Reserved_Bit15							:=	gu16_OrionBMS1_DTC_Flags1.15;

OrionBMS1_DTCFlags2_0A1F_InternalCommunicationFault			:=	gu16_OrionBMS1_DTC_Flags2.0;
OrionBMS1_DTCFlags2_0A12_CellBalancingStruckOffFault		:=	gu16_OrionBMS1_DTC_Flags2.1;
OrionBMS1_DTCFlags2_0A80_WeakCellFault						:=	gu16_OrionBMS1_DTC_Flags2.2;
OrionBMS1_DTCFlags2_0AFA_LowCellVoltageFault				:=	gu16_OrionBMS1_DTC_Flags2.3;
OrionBMS1_DTCFlags2_0A04_OpenWiringFault					:=	gu16_OrionBMS1_DTC_Flags2.4;
OrionBMS1_DTCFlags2_0AC0_CurrentSensorFault					:=	gu16_OrionBMS1_DTC_Flags2.5;
OrionBMS1_DTCFlags2_0A0D_HighestCellVoltageOver5vFault		:=	gu16_OrionBMS1_DTC_Flags2.6;
OrionBMS1_DTCFlags2_0A0F_CellASICFault						:=	gu16_OrionBMS1_DTC_Flags2.7;
OrionBMS1_DTCFlags2_0A02_WeakPackFault						:=	gu16_OrionBMS1_DTC_Flags2.8;
OrionBMS1_DTCFlags2_0A81_FanMonitorFault					:=	gu16_OrionBMS1_DTC_Flags2.9;
OrionBMS1_DTCFlags2_0A9C_ThermistorFault					:=	gu16_OrionBMS1_DTC_Flags2.10;
OrionBMS1_DTCFlags2_0100_ExternalCommunicationFault			:=	gu16_OrionBMS1_DTC_Flags2.11;
OrionBMS1_DTCFlags2_0560_RedundantPowerSupplyFault			:=	gu16_OrionBMS1_DTC_Flags2.12;
OrionBMS1_DTCFlags2_0AA6_HighVoltageIsolatonFault			:=	gu16_OrionBMS1_DTC_Flags2.13;
OrionBMS1_DTCFlags2_0A05_InputPowerSupplyFault				:=	gu16_OrionBMS1_DTC_Flags2.14;
OrionBMS1_DTCFlags2_0A06_ChargeLimitEnforcementFault		:=	gu16_OrionBMS1_DTC_Flags2.15;

gq_BMS1_BalActive			:=	gu8_OrionBMS1_Custom_Flag_1.0;
gq_BMS1_Flag_1				:=	gu8_OrionBMS1_Custom_Flag_1.1;
gq_BMS1_Flag_2				:=	gu8_OrionBMS1_Custom_Flag_1.2;
gq_BMS1_Flag_3				:=	gu8_OrionBMS1_Custom_Flag_1.3;
gq_BMS1_Flag_4				:=	gu8_OrionBMS1_Custom_Flag_1.4;
gq_BMS1_Flag_5				:=	gu8_OrionBMS1_Custom_Flag_1.5;
gq_BMS1_Flag_6				:=	gu8_OrionBMS1_Custom_Flag_1.6;
Safety_OK    				:=	gu8_OrionBMS2_Custom_Flag_1.7;

END_PROGRAM

// Application/UserCode/BMS/OrionBMS/OrionBMS2_Rx
PROGRAM OrionBMS2_Rx
VAR
	OrionBMS2_6B0_Rx	:	Receive_CAN3_STD;
	OrionBMS2_6B1_Rx	:	Receive_CAN3_STD;
	OrionBMS2_6B2_Rx	:	Receive_CAN3_STD;
	OrionBMS2_6B3_Rx	:	Receive_CAN3_STD;
	OrionBMS2_6B4_Rx	:	Receive_CAN3_STD;
	OrionBMS2_6B5_Rx	:	Receive_CAN3_STD;
	OrionBMS2_6B6_Rx	:	Receive_CAN3_STD;
	OrionBMS2_6B7_Rx	:	Receive_CAN3_STD;
	OrionBMS2_6B8_Rx	:	Receive_CAN3_STD;
	OrionBMS2_6B9_Rx	:	Receive_CAN3_STD;
	OrionBMS2_6BA_Rx	:	Receive_CAN3_STD;
	OrionBMS2_6BB_Rx	:	Receive_CAN3_STD;
	OrionBMS2_6BC_Rx	:	Receive_CAN3_STD;
	OrionBMS2_6BD_Rx	:	Receive_CAN3_STD;
	
	OrionBMS2_6B0_Rx_Timer	:	TON;
	OrionBMS2_6B1_Rx_Timer	:	TON;
	OrionBMS2_6B2_Rx_Timer	:	TON;
	OrionBMS2_6B3_Rx_Timer	:	TON;
	OrionBMS2_6B4_Rx_Timer	:	TON;
	OrionBMS2_6B5_Rx_Timer	:	TON;
	OrionBMS2_6B6_Rx_Timer	:	TON;
	OrionBMS2_6B7_Rx_Timer	:	TON;
	OrionBMS2_6B8_Rx_Timer	:	TON;
	OrionBMS2_6B9_Rx_Timer	:	TON;
	OrionBMS2_6BA_Rx_Timer	:	TON;
	OrionBMS2_6BB_Rx_Timer	:	TON;
	OrionBMS2_6BC_Rx_Timer	:	TON;
	OrionBMS2_6BD_Rx_Timer	:	TON;
	END_VAR

(*Program to receive all data from the Orion BMS*)
(*Initial saving CAN messages to receipt strucutres*)
OrionBMS2_6B0_Rx(u32_COBID	:=	16#6B0,
				 q_NewData => ,
				 au8_Data => ,
				 u8_Length => 			);
				 
OrionBMS2_6B1_Rx(u32_COBID	:=	16#6B1,
				 q_NewData => ,
				 au8_Data => ,
				 u8_Length => 			);
				 
OrionBMS2_6B2_Rx(u32_COBID	:=	16#6B2,
				 q_NewData => ,
				 au8_Data => ,
				 u8_Length => 			);
				 
OrionBMS2_6B3_Rx(u32_COBID	:=	16#6B3,
				 q_NewData => ,
				 au8_Data => ,
				 u8_Length => 			);
				 
OrionBMS2_6B4_Rx(u32_COBID	:=	16#6B4,
				 q_NewData => ,
				 au8_Data => ,
				 u8_Length => 			);
				 
OrionBMS2_6B5_Rx(u32_COBID	:=	16#6B5,
				 q_NewData => ,
				 au8_Data => ,
				 u8_Length => 			);
				 
OrionBMS2_6B6_Rx(u32_COBID	:=	16#6B6,
				 q_NewData => ,
				 au8_Data => ,
				 u8_Length => 			);
				 
OrionBMS2_6B7_Rx(u32_COBID	:=	16#6B7,
				 q_NewData => ,
				 au8_Data => ,
				 u8_Length => 			);
			 
OrionBMS2_6B8_Rx(u32_COBID	:=	16#6B8,
				 q_NewData => ,
				 au8_Data => ,
				 u8_Length => 			);
				 
OrionBMS2_6B9_Rx(u32_COBID	:=	16#6B9,
				 q_NewData => ,
				 au8_Data => ,
				 u8_Length => 			);
				 
OrionBMS2_6BA_Rx(u32_COBID	:=	16#6BA,
				 q_NewData => ,
				 au8_Data => ,
				 u8_Length => 			);
				 
OrionBMS2_6BB_Rx(u32_COBID	:=	16#6BB,
				 q_NewData => ,
				 au8_Data => ,
				 u8_Length => 			);
				 
OrionBMS2_6BC_Rx(u32_COBID	:=	16#6BC,
				 q_NewData => ,
				 au8_Data => ,
				 u8_Length => 			);
				 
OrionBMS2_6BD_Rx(u32_COBID	:=	16#6BD,
				 q_NewData => ,
				 au8_Data => ,
				 u8_Length => 			);


(*Unpacking input structures into variables*)
(*6B0*)

gs16_OrionBMS2_PackCurrent	:=	USINT_TO_INT(OrionBMS2_6B0_Rx.au8_Data[0]) +
								SHL(USINT_TO_INT(OrionBMS2_6B0_Rx.au8_Data[1]), 8);
gu16_OrionBMS2_PackVoltage	:=	USINT_TO_UINT(OrionBMS2_6B0_Rx.au8_Data[2]) +
								SHL(USINT_TO_UINT(OrionBMS2_6B0_Rx.au8_Data[3]), 8);
gu8_OrionBMS2_RAW_SOC	:=	OrionBMS2_6B0_Rx.au8_Data[4];
gu16_OrionBMS2_RelayState	:=	USINT_TO_UINT(OrionBMS2_6B0_Rx.au8_Data[5]) +
								SHL(USINT_TO_UINT(OrionBMS2_6B0_Rx.au8_Data[6]), 8);
gu8_OrionBMS2_Custom_Flag_1	:=	OrionBMS2_6B0_Rx.au8_Data[7];

(*6B1*)
gu8_OrionBMS2_Isolation_ADC			:=	USINT_TO_UINT(OrionBMS2_6B1_Rx.au8_Data[0]) +
									SHL(USINT_TO_UINT(OrionBMS2_6B1_Rx.au8_Data[1]), 8);
gu8_OrionBMS2_Shortest_Wave			:=	USINT_TO_UINT(OrionBMS2_6B1_Rx.au8_Data[2]) +
									SHL(USINT_TO_UINT(OrionBMS2_6B1_Rx.au8_Data[3]), 8);
gu16_OrionBMS2_Isolation_Clipping	:=	USINT_TO_UINT(OrionBMS2_6B1_Rx.au8_Data[4]) +
									SHL(USINT_TO_UINT(OrionBMS2_6B1_Rx.au8_Data[5]), 8);
gu16_OrionBMS2_Isolation_Threshold	:=	USINT_TO_UINT(OrionBMS2_6B1_Rx.au8_Data[6]) +
									SHL(USINT_TO_UINT(OrionBMS2_6B1_Rx.au8_Data[7]), 8);
									
(*6B2*)
gu16_OrionBMS2_DTC_Flags1		:=	USINT_TO_UINT(OrionBMS2_6B2_Rx.au8_Data[0]) +
								SHL(USINT_TO_UINT(OrionBMS2_6B2_Rx.au8_Data[1]), 8);
gu16_OrionBMS2_DTC_Flags2		:=	USINT_TO_UINT(OrionBMS2_6B2_Rx.au8_Data[2]) +
								SHL(USINT_TO_UINT(OrionBMS2_6B2_Rx.au8_Data[3]), 8);
gu16_OrionBMS2_FailsafeStatus	:=	USINT_TO_UINT(OrionBMS2_6B2_Rx.au8_Data[4]) +
								SHL(USINT_TO_UINT(OrionBMS2_6B2_Rx.au8_Data[5]), 8);
gu16_OrionBMS2_CurrentLimit		:=	USINT_TO_UINT(OrionBMS2_6B2_Rx.au8_Data[6]) +
								SHL(USINT_TO_UINT(OrionBMS2_6B2_Rx.au8_Data[7]), 8);
(*6B3*)
gu8_OrionBMS2_PackHealth			:=	OrionBMS2_6B3_Rx.au8_Data[0];
gu16_OrionBMS2_PackCycles			:=	USINT_TO_UINT(OrionBMS2_6B3_Rx.au8_Data[1]) +
									SHL(USINT_TO_UINT(OrionBMS2_6B3_Rx.au8_Data[2]), 8);
gu16_OrionBMS2_PackResistance		:=	USINT_TO_UINT(OrionBMS2_6B3_Rx.au8_Data[3]) +
									SHL(USINT_TO_UINT(OrionBMS2_6B3_Rx.au8_Data[4]), 8);
gu8_OrionBMS2_PopulatedCells		:=	OrionBMS2_6B3_Rx.au8_Data[5];
gu16_OrionBMS2_MaximumPackVoltage	:=	USINT_TO_UINT (OrionBMS2_6B3_Rx.au8_Data[6]) +
									SHL(USINT_TO_UINT(OrionBMS2_6B3_Rx.au8_Data[7]),8);

(*6B4*)
gu8_OrionBMS2_HighTemp		:=	OrionBMS2_6B4_Rx.au8_Data[0];
gu8_OrionBMS2_LowTemp		:=	OrionBMS2_6B4_Rx.au8_Data[1];
gu8_OrionBMS2_AverageTemp	:=	OrionBMS2_6B4_Rx.au8_Data[2];
gu8_OrionBMS2_InternalTemp	:=	OrionBMS2_6B4_Rx.au8_Data[3];
gu16_OrionBMS2_MinimumPackVoltage	:=	USINT_TO_UINT(OrionBMS2_6B4_Rx.au8_Data[4]) +
									SHL(USINT_TO_UINT(OrionBMS2_6B4_Rx.au8_Data[5]), 8);
gu16_OrionBMS2_PackAmphours	:=	USINT_TO_UINT(OrionBMS2_6B4_Rx.au8_Data[6]) +
								SHL(USINT_TO_UINT(OrionBMS2_6B4_Rx.au8_Data[7]), 8);
(*6B5*)
gu16_OrionBMS2_AverageCellVoltage	:=	USINT_TO_UINT(OrionBMS2_6B5_Rx.au8_Data[0]) +
										SHL(USINT_TO_UINT(OrionBMS2_6B5_Rx.au8_Data[1]), 8);
gu16_OrionBMS2_LowCellVoltage		:=	USINT_TO_UINT(OrionBMS2_6B5_Rx.au8_Data[2]) +
										SHL(USINT_TO_UINT(OrionBMS2_6B5_Rx.au8_Data[3]), 8);
gu16_OrionBMS2_HighCellVoltage		:=	USINT_TO_UINT(OrionBMS2_6B5_Rx.au8_Data[4]) +
										SHL(USINT_TO_UINT(OrionBMS2_6B5_Rx.au8_Data[5]), 8);
gu8_OrionBMS2_LowCellVoltNumber		:=	OrionBMS2_6B5_Rx.au8_Data[6];
gu8_OrionBMS2_HighCellVoltNumber	:=	OrionBMS2_6B5_Rx.au8_Data[7];
(*6B6*)
gu8_OrionBMS2_Low_Intres_ID			:=	OrionBMS2_6B6_Rx.au8_Data[0];
gu8_OrionBMS2_High_Intres_ID		:=	OrionBMS2_6B6_Rx.au8_Data[1];
gu16_OrionBMS2_Low_Cell_Resistance	:=	USINT_TO_UINT(OrionBMS2_6B6_Rx.au8_Data[2]) +
										SHL(USINT_TO_UINT(OrionBMS2_6B6_Rx.au8_Data[3]), 8);
gu16_OrionBMS2_High_Cell_Resistance	:=	USINT_TO_UINT(OrionBMS2_6B6_Rx.au8_Data[4]) +
										SHL(USINT_TO_UINT(OrionBMS2_6B6_Rx.au8_Data[5]), 8);
gu16_OrionBMS2_Average_Cell_Resistance	:=	USINT_TO_UINT(OrionBMS2_6B6_Rx.au8_Data[6]) +
										SHL(USINT_TO_UINT(OrionBMS2_6B6_Rx.au8_Data[7]), 8);

(*6B7*)
gu8_OrionBMS2_Low_Thermistor_ID			:=	OrionBMS2_6B7_Rx.au8_Data[0];
gu8_OrionBMS2_High_Thermistor_ID		:=	OrionBMS2_6B7_Rx.au8_Data[1];
gu16_OrionBMS2_PackDCL				:=	USINT_TO_UINT(OrionBMS2_6B7_Rx.au8_Data[2]) +
										SHL(USINT_TO_UINT(OrionBMS2_6B7_Rx.au8_Data[3]), 8);
gu16_OrionBMS2_PackCCL				:=	USINT_TO_UINT(OrionBMS2_6B7_Rx.au8_Data[4]) +
										SHL(USINT_TO_UINT(OrionBMS2_6B7_Rx.au8_Data[5]), 8);
gu16_OrionBMS2_PackSummedVoltage	:=	USINT_TO_UINT(OrionBMS2_6B7_Rx.au8_Data[6]) +
										SHL(USINT_TO_UINT(OrionBMS2_6B7_Rx.au8_Data[7]), 8);

(*6B8*)
	gu8_OrionBMS2_Firmware_Minor	:=	OrionBMS2_6B8_Rx.au8_Data[0];	
	gu8_OrionBMS2_Firmware_Patch	:=	OrionBMS2_6B8_Rx.au8_Data[1];		
	gu8_OrionBMS2_Constant_2		:=	OrionBMS2_6B8_Rx.au8_Data[2];		
	gu8_OrionBMS2_Constant_3		:=	OrionBMS2_6B8_Rx.au8_Data[3];		
	gu8_OrionBMS2_Constant_4		:=	OrionBMS2_6B8_Rx.au8_Data[4];		
	gu16_OrionBMS2_CheckSum			:=	USINT_TO_UINT(OrionBMS2_6B8_Rx.au8_Data[5]) +
										SHL(USINT_TO_UINT(OrionBMS2_6B8_Rx.au8_Data[6]), 8);
	gu8_OrionBMS2_Spare_6B6_7	:=	OrionBMS2_6B8_Rx.au8_Data[7];


(*6B9*)
gu8_OrionBMS2_6B9_0		:=	OrionBMS2_6B9_Rx.au8_Data[0];
gu8_OrionBMS2_6B9_1		:=	OrionBMS2_6B9_Rx.au8_Data[1];
gu8_OrionBMS2_6B9_2		:=	OrionBMS2_6B9_Rx.au8_Data[2];
gu8_OrionBMS2_6B9_3		:=	OrionBMS2_6B9_Rx.au8_Data[3];
gu8_OrionBMS2_6B9_4		:=	OrionBMS2_6B9_Rx.au8_Data[4];
gu8_OrionBMS2_6B9_5		:=	OrionBMS2_6B9_Rx.au8_Data[5];
gu8_OrionBMS2_6B9_6		:=	OrionBMS2_6B9_Rx.au8_Data[6];
gu8_OrionBMS2_6B9_7		:=	OrionBMS2_6B9_Rx.au8_Data[7];


(*6BA*)
gu8_OrionBMS2_6BA_0		:=	OrionBMS2_6BA_Rx.au8_Data[0];
gu8_OrionBMS2_6BA_1		:=	OrionBMS2_6BA_Rx.au8_Data[1];
gu8_OrionBMS2_6BA_2		:=	OrionBMS2_6BA_Rx.au8_Data[2];
gu8_OrionBMS2_6BA_3		:=	OrionBMS2_6BA_Rx.au8_Data[3];
gu8_OrionBMS2_6BA_4		:=	OrionBMS2_6BA_Rx.au8_Data[4];
gu8_OrionBMS2_6BA_5		:=	OrionBMS2_6BA_Rx.au8_Data[5];
gu8_OrionBMS2_6BA_6		:=	OrionBMS2_6BA_Rx.au8_Data[6];
gu8_OrionBMS2_6BA_7		:=	OrionBMS2_6BA_Rx.au8_Data[7];

(*6BB*)
gu8_OrionBMS2_6BB_0		:=	OrionBMS2_6BB_Rx.au8_Data[0];
gu8_OrionBMS2_6BB_1		:=	OrionBMS2_6BB_Rx.au8_Data[1];
gu8_OrionBMS2_6BB_2		:=	OrionBMS2_6BB_Rx.au8_Data[2];
gu8_OrionBMS2_6BB_3		:=	OrionBMS2_6BB_Rx.au8_Data[3];
gu8_OrionBMS2_6BB_4		:=	OrionBMS2_6BB_Rx.au8_Data[4];
gu8_OrionBMS2_6BB_5		:=	OrionBMS2_6BB_Rx.au8_Data[5];
gu8_OrionBMS2_6BB_6		:=	OrionBMS2_6BB_Rx.au8_Data[6];
gu8_OrionBMS2_6BB_7		:=	OrionBMS2_6BB_Rx.au8_Data[7];

(*6BC*)
gu8_OrionBMS2_6BC_0		:=	OrionBMS2_6BC_Rx.au8_Data[0];
gu8_OrionBMS2_6BC_1		:=	OrionBMS2_6BC_Rx.au8_Data[1];
gu8_OrionBMS2_6BC_2		:=	OrionBMS2_6BC_Rx.au8_Data[2];
gu8_OrionBMS2_6BC_3		:=	OrionBMS2_6BC_Rx.au8_Data[3];
gu8_OrionBMS2_6BC_4		:=	OrionBMS2_6BC_Rx.au8_Data[4];
gu8_OrionBMS2_6BC_5		:=	OrionBMS2_6BC_Rx.au8_Data[5];
gu8_OrionBMS2_6BC_6		:=	OrionBMS2_6BC_Rx.au8_Data[6];
gu8_OrionBMS2_6BC_7		:=	OrionBMS2_6BC_Rx.au8_Data[7];	
	
(*6BD*)
gu8_OrionBMS2_6BD_0		:=	OrionBMS2_6BD_Rx.au8_Data[0];
gu8_OrionBMS2_6BD_1		:=	OrionBMS2_6BD_Rx.au8_Data[1];
gu8_OrionBMS2_6BD_2		:=	OrionBMS2_6BD_Rx.au8_Data[2];
gu8_OrionBMS2_6BD_3		:=	OrionBMS2_6BD_Rx.au8_Data[3];
gu8_OrionBMS2_6BD_4		:=	OrionBMS2_6BD_Rx.au8_Data[4];
gu8_OrionBMS2_6BD_5		:=	OrionBMS2_6BD_Rx.au8_Data[5];
gu8_OrionBMS2_6BD_6		:=	OrionBMS2_6BD_Rx.au8_Data[6];
gu8_OrionBMS2_6BD_7		:=	OrionBMS2_6BD_Rx.au8_Data[7];


(*Communications loss check*)
OrionBMS2_6B0_Rx_Timer(IN := NOT(OrionBMS2_6B0_Rx.q_NewData), PT := T#3S);
OrionBMS2_6B1_Rx_Timer(IN := NOT(OrionBMS2_6B1_Rx.q_NewData), PT := T#3S);
OrionBMS2_6B2_Rx_Timer(IN := NOT(OrionBMS2_6B2_Rx.q_NewData), PT := T#3S);
OrionBMS2_6B3_Rx_Timer(IN := NOT(OrionBMS2_6B3_Rx.q_NewData), PT := T#3S);
OrionBMS2_6B4_Rx_Timer(IN := NOT(OrionBMS2_6B4_Rx.q_NewData), PT := T#3S);
OrionBMS2_6B5_Rx_Timer(IN := NOT(OrionBMS2_6B5_Rx.q_NewData), PT := T#3S);
OrionBMS2_6B6_Rx_Timer(IN := NOT(OrionBMS2_6B6_Rx.q_NewData), PT := T#3S);
OrionBMS2_6B7_Rx_Timer(IN := NOT(OrionBMS2_6B7_Rx.q_NewData), PT := T#3S);
OrionBMS2_6B8_Rx_Timer(IN := NOT(OrionBMS2_6B8_Rx.q_NewData), PT := T#3S);
OrionBMS2_6B9_Rx_Timer(IN := NOT(OrionBMS2_6B9_Rx.q_NewData), PT := T#3S);
OrionBMS2_6BA_Rx_Timer(IN := NOT(OrionBMS2_6BA_Rx.q_NewData), PT := T#3S);
OrionBMS2_6BB_Rx_Timer(IN := NOT(OrionBMS2_6BB_Rx.q_NewData), PT := T#3S);
OrionBMS2_6BC_Rx_Timer(IN := NOT(OrionBMS2_6BC_Rx.q_NewData), PT := T#3S);
OrionBMS2_6BD_Rx_Timer(IN := NOT(OrionBMS2_6BD_Rx.q_NewData), PT := T#3S);
IF (OrionBMS2_6B0_Rx_Timer.Q = TRUE AND OrionBMS2_6B1_Rx_Timer.Q = TRUE AND OrionBMS2_6B2_Rx_Timer.Q = TRUE AND
	OrionBMS2_6B3_Rx_Timer.Q = TRUE AND OrionBMS2_6B4_Rx_Timer.Q = TRUE AND OrionBMS2_6B5_Rx_Timer.Q = TRUE AND
	OrionBMS2_6B6_Rx_Timer.Q = TRUE AND OrionBMS2_6B7_Rx_Timer.Q = TRUE AND OrionBMS2_6B8_Rx_Timer.Q = TRUE AND
	OrionBMS2_6B9_Rx_Timer.Q = TRUE AND OrionBMS2_6BA_Rx_Timer.Q = TRUE AND OrionBMS2_6BB_Rx_Timer.Q = TRUE AND
	OrionBMS2_6BC_Rx_Timer.Q = TRUE AND OrionBMS2_6BD_Rx_Timer.Q = TRUE											) THEN

	gq_OrionBMS2_CommsLoss	:=	TRUE;
ELSE
	gq_OrionBMS2_CommsLoss	:=	FALSE;
END_IF


OrionBMS2_RxConversion();

END_PROGRAM

// Application/UserCode/BELDCDC/BELDCDC_Rx
PROGRAM BELDCDC_Rx
VAR
	BelDCDC_FWS_Rx	:	Receive_CAN1_EXD;
	BelDCDC_IO_Rx	:	Receive_CAN1_EXD;
	
	BelDCDC_FWS_Rx_Timer	:	TON;
	BelDCDC_IO_Rx_Timer		:	TON;
	hton_Startup_Timer		:	TON;
END_VAR

(*Message receipt for the DCDCs*)

(*Receive the messages from the DCDC*)
BelDCDC_FWS_Rx(u32_COBID	:=	16#18FFD4B3,
				 q_NewData => ,
				 au8_Data => ,
				 u8_Length => 			);

BelDCDC_IO_Rx(u32_COBID	:=	16#18FFD6B3,
				 q_NewData => ,
				 au8_Data => ,
				 u8_Length => 			);

(*Wait an initial time from when the DCDC is switched on to prevent falsly detecting faults*)
hton_Startup_Timer(IN := DO_q_DrivetrainDCDCInhibit_DO, PT := T#1000MS);
IF (hton_Startup_Timer.Q = TRUE) THEN (*During startup errors are reported while precharge occurs so this ignores the initiall error reporting*)
	gq_BelDCDC_flt_InputUV			:=	BelDCDC_FWS_Rx.au8_Data[0].0;
	gq_BelDCDC_flt_InputOV			:=	BelDCDC_FWS_Rx.au8_Data[0].1;
	gq_BelDCDC_flt_OutputUV			:=	BelDCDC_FWS_Rx.au8_Data[0].2;
	gq_BelDCDC_flt_OutputOV			:=	BelDCDC_FWS_Rx.au8_Data[0].3;
	gq_BelDCDC_flt_OutputOC			:=	BelDCDC_FWS_Rx.au8_Data[0].4;
	gq_BelDCDC_flt_OTP				:=	BelDCDC_FWS_Rx.au8_Data[0].5;
	gq_BelDCDC_flt_I2CFault			:=	BelDCDC_FWS_Rx.au8_Data[0].6;
	gq_BelDCDC_flt_CANFault			:=	BelDCDC_FWS_Rx.au8_Data[0].7;
	gq_BelDCDC_flt_EEPROM_CRCFault	:=	BelDCDC_FWS_Rx.au8_Data[1].0;
	gq_BelDCDC_flt_ShortCircuit		:=	BelDCDC_FWS_Rx.au8_Data[1].1;
	gq_BelDCDC_flt_ThermistorFault	:=	BelDCDC_FWS_Rx.au8_Data[1].2;
	gq_BelDCDC_flt_Overload			:=	BelDCDC_FWS_Rx.au8_Data[1].3;
	gq_BelDCDC_flt_OutputOVLatch	:=	BelDCDC_FWS_Rx.au8_Data[1].4;
	gq_BelDCDC_flt_ReversePolarity	:=	BelDCDC_FWS_Rx.au8_Data[1].5;
	gq_BelDCDC_war_CoolantOTP		:=	BelDCDC_FWS_Rx.au8_Data[3].0;
	gq_BelDCDC_war_CurrentLimiting	:=	BelDCDC_FWS_Rx.au8_Data[3].1;
	gq_BelDCDC_sts_UnitEnabled		:=	BelDCDC_FWS_Rx.au8_Data[6].0;
	gq_BelDCDC_sts_Wakeup			:=	BelDCDC_FWS_Rx.au8_Data[6].1;
	gq_BelDCDC_sts_Fault			:=	BelDCDC_FWS_Rx.au8_Data[6].2;
	gq_BelDCDC_sts_LatchedFault		:=	BelDCDC_FWS_Rx.au8_Data[6].3;
	gq_BelDCDC_sts_RemoteShutdown	:=	BelDCDC_FWS_Rx.au8_Data[6].4;
	gq_BelDCDC_sts_StartupInitDone	:=	BelDCDC_FWS_Rx.au8_Data[6].5;
	gq_BelDCDC_sts_InputOK			:=	BelDCDC_FWS_Rx.au8_Data[6].6;
	gq_BelDCDC_sts_HVILOK			:=	BelDCDC_FWS_Rx.au8_Data[6].7;
	gq_BelDCDC_sts_ReversePolarity	:=	BelDCDC_FWS_Rx.au8_Data[7].0;
	gq_BelDCDC_sts_Hiccup			:=	BelDCDC_FWS_Rx.au8_Data[7].1;
END_IF
(*IO*)
gu16_BelDCDC_OutputVoltage_Rx	:=	USINT_TO_UINT(BelDCDC_IO_Rx.au8_Data[0]) +
									SHL(USINT_TO_UINT(BelDCDC_IO_Rx.au8_Data[1]), 8);
gu16_BelDCDC_OutputCurrent_Rx	:=	USINT_TO_UINT(BelDCDC_IO_Rx.au8_Data[2]) +
									SHL(USINT_TO_UINT(BelDCDC_IO_Rx.au8_Data[3]), 8);
gu16_BelDCDC_InputVoltage_Rx	:=	USINT_TO_UINT(BelDCDC_IO_Rx.au8_Data[4]) +
									SHL(USINT_TO_UINT(BelDCDC_IO_Rx.au8_Data[5]), 8);
gu16_BelDCDC_TempCoolant_Rx		:=	USINT_TO_UINT(BelDCDC_IO_Rx.au8_Data[6]) +
									SHL(USINT_TO_UINT(BelDCDC_IO_Rx.au8_Data[7]), 8);

(*Bel DCDC only seems to send messages on startup*)
(*When the output is set then detect if messages are being sent if no message is received for 5 seconds then report a communications loss*)
BelDCDC_FWS_Rx_Timer(IN := (NOT(BelDCDC_FWS_Rx.q_NewData) AND DO_q_DrivetrainDCDCInhibit_DO = TRUE), PT := T#5S);
BelDCDC_IO_Rx_Timer(IN := (NOT(BelDCDC_IO_Rx.q_NewData) AND DO_q_DrivetrainDCDCInhibit_DO = TRUE), PT := T#5S);
IF (BelDCDC_FWS_Rx_Timer.Q = TRUE AND BelDCDC_IO_Rx_Timer.Q = TRUE) THEN
	gq_BELDCDC_CommsLoss	:=	TRUE;
ELSE
	gq_BELDCDC_CommsLoss	:=	FALSE;
END_IF									

BELDCDC_RxConversion();

END_PROGRAM

// Application/UserCode/BELDCDC/BELDCDC_RxConversion
PROGRAM BELDCDC_RxConversion
VAR
END_VAR

(*Take the values received on CANbus and apply the offset and conversion factor to each where necessary*)
gr_BelDCDC_OutputVoltage		:=	UINT_TO_REAL(gu16_BelDCDC_OutputVoltage_Rx) * 0.05;
gr_BelDCDC_OutputCurrent		:=	UINT_TO_REAL(gu16_BelDCDC_OutputCurrent_Rx) * 0.05;
gr_BelDCDC_InputVoltage			:=	UINT_TO_REAL(gu16_BelDCDC_InputVoltage_Rx) * 0.05;
gr_BelDCDC_TempCoolant			:=	UINT_TO_REAL(gu16_BelDCDC_TempCoolant_Rx) * 0.1;

END_PROGRAM

// Application/UserCode/CAN Function Blocks/CAN1/Receive_CAN1_EXD
FUNCTION_BLOCK Receive_CAN1_EXD
VAR_INPUT
	u32_COBID	:	DWORD;
END_VAR
VAR_OUTPUT
	q_NewData	:	BOOL;
	au8_Data	:	ARRAY [0..7] OF BYTE;
	u8_Length	:	BYTE;
END_VAR
VAR
	hq_Initialise	:	BOOL	:=	FALSE;
	ht_RxMessage	:	t_CANReceive;
	ht_MsgRx		:	Callback_Receive_CAN1;
END_VAR



IF (hq_Initialise = FALSE) THEN
	(*
	(*11 bit*)
	G_CAN1_Channel.AddCOBID(i_CobId := u32_COBID,
							i_itfCallback := ht_RxMessage,
							i_Argument := ADR(ht_RxMessage));
	*)
	(*29 bit*)
	G_CAN1_Channel.AddCOBID(i_CobId := u32_COBID OR EPEC_CANVXD.MASK_29BIT,
							i_itfCallback := ht_MsgRx,
							i_Argument := ADR(ht_RxMessage));
	G_CAN1_Channel.SetMask(i_CobID := u32_COBID OR EPEC_CANVXD.MASK_29BIT, i_Mask := (*16#0CFF0211 OR 16#0C010305 OR*) EPEC_CANVXD.MASK_29BIT);

	hq_Initialise	:=	TRUE;
END_IF


IF (ht_RxMessage.q_NewDataRxed = TRUE) THEN
	au8_Data	:=	ht_RxMessage.Data;
	u8_Length	:=	ht_RxMessage.Len;
	q_NewData	:=	TRUE;
	ht_RxMessage.q_NewDataRxed	:=	FALSE;
ELSE
	q_NewData	:=	FALSE;
END_IF

END_FUNCTION_BLOCK

// Application/UserCode/BELDCDC/BELDCDC_Tx
PROGRAM BELDCDC_Tx
VAR
	
	BelDCDC_TX				:	EPEC_CANVXD.Msg;
	hton_MessageSend_Timer	:	TON;
	// Enable Bit (There is also a HW wire)
	DCDC_Enable: BYTE := 1;
END_VAR

(*Message Transmit for the DCDC*)
BelDCDC_TX.ID	:=	16#18EFB300 OR EPEC_CANVXD.MASK_29BIT;//* message to control DCDC
BelDCDC_TX.Data[0]	:=	0;//* system requirement.
BelDCDC_TX.Data[1]	:=	WORD_TO_BYTE (BELDCDC_TxConversion.RAW_DCDC_Voltage_SP);//*LSB
BelDCDC_TX.Data[2]	:=	WORD_TO_BYTE (SHR (BELDCDC_TxConversion.RAW_DCDC_Voltage_SP,8));//*MSB
BelDCDC_TX.Data[3]	:=	WORD_TO_BYTE (BELDCDC_TxConversion.RAW_DCDC_Current_SP);//*LSB
BelDCDC_TX.Data[4]	:=	WORD_TO_BYTE (SHR (BELDCDC_TxConversion.RAW_DCDC_Current_SP,8));//*MSB
BelDCDC_TX.Data[5]	:=	DCDC_Enable;
BelDCDC_TX.Data[6]	:=	255;//* system requirement.
BelDCDC_TX.Data[7]	:=	255;//* system requirement.
BelDCDC_TX.Len		:=	8;


hton_MessageSend_Timer(IN := NOT(hton_MessageSend_Timer.Q), PT := T#200MS);//* Tx every 200ms
IF (hton_MessageSend_Timer.Q = TRUE) THEN
G_CAN1_Channel.SendMessage(i_pMSG:=ADR(BelDCDC_TX));
END_IF

END_PROGRAM

// Application/UserCode/BELDCDC/BELDCDC_TxConversion
PROGRAM BELDCDC_TxConversion
VAR
	RAW_DCDC_Voltage_SP: WORD;
	RAW_DCDC_Current_SP: WORD;
	// Amperage
	DCDC_Current_SP: REAL := 100;
	// Battery Voltage
	DCDC_Voltage_SP: REAL :=27.6;	
END_VAR

(*Take the values and Tx over CANbus and apply the offset and conversion factor to each where necessary*)

RAW_DCDC_Voltage_SP					:=REAL_TO_WORD(DCDC_Voltage_SP*20);
RAW_DCDC_Current_SP					:=REAL_TO_WORD (DCDC_Current_SP*20);

END_PROGRAM

// Application/UserCode/CAN1/CAN1_Rx
PROGRAM CAN1_Rx
VAR
	Accelerator_Dennis_Rx	:	Receive_CAN1_EXD_28bit;
	Brake_Dennis_Rx			:	Receive_CAN1_EXD;
	GearSelect_Dennis_Rx	:	Receive_CAN1_EXD_28bit;
	AirPressure_Dennis_Rx	:	Receive_CAN1_EXD;
	
	EBC1_KB_Rx				:	Receive_CAN1_EXD;
	VDC1_KB_Rx				:	Receive_CAN1_EXD;
	EBC2_KB_Rx				:	Receive_CAN1_EXD;
	
	RegenStick01_Rx			:	Receive_CAN1_EXD;
	RegenStick12_Rx			:	Receive_CAN1_EXD;
	
	Bob_Handbrake_Rx	:	Receive_CAN1_EXD;
	Bob_Brake_Rx		:	Receive_CAN1_EXD;
	Bob_Accel_Rx		:	Receive_CAN1_EXD;
	Bob_RegenSelector_Rx	:	Receive_CAN1_EXD;
	
	Bob_WheelSpeed_Rx	:	Receive_CAN1_EXD_28bit;
	Bob_J1939_AirPressure_Rx	:	Receive_CAN1_EXD;
	
	Temperature_Rx		:	Receive_CAN1_EXD;
	Dennis_StabTracDisable_Rx	:	Receive_CAN1_EXD;
	
	Accelerator_Dennis_Rx_Timer	:	TON;
	Brake_Dennis_Rx_Timer		:	TON;
	GearSelect_Dennis_Rx_Timer	:	TON;
	Airpressure_Dennis_Rx_Timer	:	TON;
	
	hq_Bob_RightDrive_Compromised	: BOOL;
	hq_Bob_LeftDrive_Compromised	: BOOL;
	hq_Bob_RightFront_Compromised	: BOOL;
	hq_Bob_LeftFront_Compromised	: BOOL;
	
	Merc_AIR1_EAPU		:	Receive_CAN1_EXD;
	MercStalk_Rx: Receive_CAN1_EXD;
	Merc_Neutral_CAN1: BOOL := FALSE;
	Merc_Drive_CAN1: BOOL := FALSE;
	Merc_Reverse_CAN1: BOOL := FALSE;
	Dennis_No_Press: BOOL;
	Dennis_Up: BOOL;
	Dennis_Down: BOOL;
	LOADCTU: BOOL;
	InitialiseCounterValue: BYTE;
END_VAR

{region "Message Rx check"}
Accelerator_Dennis_Rx	(u32_COBID	:=	16#0CFF0211,
						q_NewData => ,
						au8_Data => ,
						u8_Length => 			);
				
(*Brake_Dennis_Rx	(u32_COBID	:=	16#18F0010B,
				q_NewData => ,
				au8_Data => ,
				u8_Length => 			);*)
				
GearSelect_Dennis_Rx	(u32_COBID	:=	16#0C010305,
						q_NewData => ,
						au8_Data => ,
						u8_Length => 			);
						
AirPressure_Dennis_Rx	(u32_COBID	:=	16#18FEAE30,
						q_NewData => ,
						au8_Data => ,
						u8_Length => 			);
						
EBC1_KB_Rx				(u32_COBID	:=	16#18F0010B,
						q_NewData => ,
						au8_Data => ,
						u8_Length => 			);

VDC1_KB_Rx				(u32_COBID	:=	16#18FE4F0B,
						q_NewData => ,
						au8_Data => ,
						u8_Length => 			);

EBC2_KB_Rx				(u32_COBID	:=	16#18FEBF0B,
						q_NewData => ,
						au8_Data => ,
						u8_Length => 			);
						
RegenStick01_Rx			(u32_COBID	:=	16#18F00021,
						q_NewData => ,
						au8_Data => ,
						u8_Length => 			);
							 
RegenStick12_Rx			(u32_COBID	:=	16#0C000003,
						q_NewData => ,
						au8_Data => ,
						u8_Length => 			);
							 
Bob_Handbrake_Rx(u32_COBID	:=	16#18FF0447,
			q_NewData => ,
			au8_Data => ,
			u8_Length => 			);
				 
Bob_Brake_Rx(u32_COBID	:=	16#14FF010B,
			q_NewData => ,
			au8_Data => ,
			u8_Length => 			);
				 
Bob_Accel_Rx(u32_COBID	:=	16#10F00300,
			q_NewData => ,
			au8_Data => ,
			u8_Length => 			);
				 
Bob_RegenSelector_Rx(u32_COBID	:=	16#14FF0300,
			q_NewData => ,
			au8_Data => ,
			u8_Length => 			);
				 
Bob_WheelSpeed_Rx(u32_COBID	:=	16#08FE6E0B,
			q_NewData => ,
			au8_Data => ,
			u8_Length => 			);
				 
Bob_J1939_AirPressure_Rx(u32_COBID := 16#14FEAE17,
			q_NewData => ,
			au8_Data => ,
			u8_Length => 			);
				 
Temperature_Rx(u32_COBID := 16#18FF12C4,
			q_NewData => ,
			au8_Data => ,
			u8_Length => 			);
				 
Dennis_StabTracDisable_Rx(u32_COBID := 16#18FE4F0B,
			q_NewData => ,
			au8_Data => ,
			u8_Length => 			);
				 
MercStalk_Rx	(u32_COBID	:=	16#18FF0400,
						q_NewData => ,
						au8_Data => ,
						u8_Length => 			);
(*Moved to CAN 3*)
Merc_AIR1_EAPU(u32_COBID := 16#14FEAE30,
		 	q_NewData => ,
			au8_Data => ,
			u8_Length =>			);			

{endregion}
Merc_Neutral_CAN1			:=	MercStalk_Rx.au8_Data[4].0;
Merc_Drive_CAN1				:=	MercStalk_Rx.au8_Data[4].1;
Merc_Reverse_CAN1			:=	MercStalk_Rx.au8_Data[4].2;
{region "Assign data to receive variables"}		
gu8_AccelPedal_Dennis_Rx	:=	Accelerator_Dennis_Rx.au8_Data[3];
gq_Dennis_Accel_NewData		:=	Accelerator_Dennis_Rx.q_NewData;				

gq_BrakePedal_Dennis_Rx		:=	Brake_Dennis_Rx.au8_Data[0].6;
gu8_BrakePedal_Perc_Dennis_Rx	:=	Brake_Dennis_Rx.au8_Data[1];

gu8_GearSelector_Dennis_Rx	:=	GearSelect_Dennis_Rx.au8_Data[2];
	 // Dennis Regen Select
		  
	InitialiseCounterValue := InitialiseCounterValue + 1;
	IF InitialiseCounterValue > 250 THEN
	InitialiseCounterValue := 201;
	END_IF
				   
 	IF GearSelect_Dennis_Rx.au8_Data[2] = 224 THEN
	Dennis_No_Press := TRUE;
	ELSE
	Dennis_No_Press := FALSE;
	END_IF
	
	IF GearSelect_Dennis_Rx.au8_Data[2] = 249 THEN
	Dennis_Up	:= TRUE;
	ELSE
	Dennis_Up := FALSE;
	END_IF
	
	IF GearSelect_Dennis_Rx.au8_Data[2] = 247 THEN
	Dennis_Down	:= TRUE;
	ELSE
	Dennis_Down := FALSE;
	END_IF
		 
	IF Dennis_Regen.DennisRegen.CV > 4 OR InitialiseCounterValue < 200 THEN 
	LOADCTU := TRUE;
	ELSE
	LOADCTU := FALSE;
	END_IF 
//		  
IF (AirPressure_Dennis_Rx.au8_Data[2] > 0 OR AirPressure_Dennis_Rx.au8_Data[3] > 0) THEN
	gu8_Dennis_AirPressureBrake1_Rx	:=	AirPressure_Dennis_Rx.au8_Data[2];
	gu8_Dennis_AirPressureBrake2_Rx	:=	AirPressure_Dennis_Rx.au8_Data[3];
	gu8_Dennis_AirPressureSusp_Rx	:=	AirPressure_Dennis_Rx.au8_Data[5];
END_IF

	 
gu8_EBC1_ASREngineControlActive				:=BOOL_TO_USINT(EBC1_KB_Rx.au8_Data[0].0) + SHL(BOOL_TO_USINT(EBC1_KB_Rx.au8_Data[0].1), 1);
gu8_EBC1_ASRBrakeControlActive				:=BOOL_TO_USINT(EBC1_KB_Rx.au8_Data[0].2) + SHL(BOOL_TO_USINT(EBC1_KB_Rx.au8_Data[0].3), 1);
gu8_EBC1_ABSActive							:=BOOL_TO_USINT(EBC1_KB_Rx.au8_Data[0].4) + SHL(BOOL_TO_USINT(EBC1_KB_Rx.au8_Data[0].5), 1);
gu8_EBC1_EBSBrakeSwitch						:=BOOL_TO_USINT(EBC1_KB_Rx.au8_Data[0].6) + SHL(BOOL_TO_USINT(EBC1_KB_Rx.au8_Data[0].7), 1);
gu8_EBC1_BrakePedalPosition					:=EBC1_KB_Rx.au8_Data[1];
gu8_EBC1_ABSOffroadSwitch					:=BOOL_TO_USINT(EBC1_KB_Rx.au8_Data[2].0) + SHL(BOOL_TO_USINT(EBC1_KB_Rx.au8_Data[2].1), 1);
gu8_EBC1_ASROffroadSwitch					:=BOOL_TO_USINT(EBC1_KB_Rx.au8_Data[2].2) + SHL(BOOL_TO_USINT(EBC1_KB_Rx.au8_Data[2].3), 1);
gu8_EBC1_ASRHillholderSwitch				:=BOOL_TO_USINT(EBC1_KB_Rx.au8_Data[2].4) + SHL(BOOL_TO_USINT(EBC1_KB_Rx.au8_Data[2].5), 1);
gu8_EBC1_TractionControlOverrideSwtich		:=BOOL_TO_USINT(EBC1_KB_Rx.au8_Data[2].6) + SHL(BOOL_TO_USINT(EBC1_KB_Rx.au8_Data[2].7), 1);
gu8_EBC1_AcceleratorInterlockSwitch			:=BOOL_TO_USINT(EBC1_KB_Rx.au8_Data[3].0) + SHL(BOOL_TO_USINT(EBC1_KB_Rx.au8_Data[3].1), 1);
gu8_EBC1_EngineDerateSwitch					:=BOOL_TO_USINT(EBC1_KB_Rx.au8_Data[3].2) + SHL(BOOL_TO_USINT(EBC1_KB_Rx.au8_Data[3].3), 1);
gu8_EBC1_EngineAuxiliaryShutdownSwitch		:=BOOL_TO_USINT(EBC1_KB_Rx.au8_Data[3].4) + SHL(BOOL_TO_USINT(EBC1_KB_Rx.au8_Data[3].5), 1);
gu8_EBC1_RemoteAcceleratorEnableSwitch		:=BOOL_TO_USINT(EBC1_KB_Rx.au8_Data[3].6) + SHL(BOOL_TO_USINT(EBC1_KB_Rx.au8_Data[3].7), 1);
gu8_EBC1_EngineRetarderSelection			:=EBC1_KB_Rx.au8_Data[4];
gu8_EBC1_ABSFullyOperational				:=BOOL_TO_USINT(EBC1_KB_Rx.au8_Data[5].0) + SHL(BOOL_TO_USINT(EBC1_KB_Rx.au8_Data[5].1), 1);
gu8_EBC1_gu8_EBC1_EBSRedWarningSignal		:=BOOL_TO_USINT(EBC1_KB_Rx.au8_Data[5].2) + SHL(BOOL_TO_USINT(EBC1_KB_Rx.au8_Data[5].3), 1);
gu8_EBC1_ABSEBSAmberWarningSignal			:=BOOL_TO_USINT(EBC1_KB_Rx.au8_Data[5].4) + SHL(BOOL_TO_USINT(EBC1_KB_Rx.au8_Data[5].5), 1);
gu8_EBC1_ATCASRInformationSignal			:=BOOL_TO_USINT(EBC1_KB_Rx.au8_Data[5].6) + SHL(BOOL_TO_USINT(EBC1_KB_Rx.au8_Data[5].7), 1);
gu8_EBC1_SrcAddrOfCrtllingDevForBrkCtrl		:=EBC1_KB_Rx.au8_Data[6];
gu8_EBC1_HaltBrakeSwitch					:=BOOL_TO_USINT(EBC1_KB_Rx.au8_Data[7].2) + SHL(BOOL_TO_USINT(EBC1_KB_Rx.au8_Data[7].3), 1);
gu8_EBC1_TrailerABSStatus					:=BOOL_TO_USINT(EBC1_KB_Rx.au8_Data[7].4) + SHL(BOOL_TO_USINT(EBC1_KB_Rx.au8_Data[7].5), 1);
gu8_EBC1_TractorMntdTrailerABSWarningSignal	:=BOOL_TO_USINT(EBC1_KB_Rx.au8_Data[7].6) + SHL(BOOL_TO_USINT(EBC1_KB_Rx.au8_Data[7].7), 1);

gu16_EBC2_KB_FrontAxleSpeed_Rx		:=	USINT_TO_UINT(EBC2_KB_Rx.au8_Data[0]) + SHL(USINT_TO_UINT(EBC2_KB_Rx.au8_Data[1]), 8);
gu16_EBC2_KB_FrontLeftRelSpd_Rx		:=	EBC2_KB_Rx.au8_Data[2];
gu16_EBC2_KB_FrontRightRelSpd_Rx	:=	EBC2_KB_Rx.au8_Data[3];
gu16_EBC2_KB_RearLeft1RelSpd_Rx		:=	EBC2_KB_Rx.au8_Data[4];
gu16_EBC2_KB_RearRight1RelSpd_Rx	:=	EBC2_KB_Rx.au8_Data[5];
gu16_EBC2_KB_RearLeft2RelSpd_Rx		:=	EBC2_KB_Rx.au8_Data[6];
gu16_EBC2_KB_RearRight2RelSpd_Rx	:=	EBC2_KB_Rx.au8_Data[7];

gu8_RegenStick01Pos					:=	RegenStick01_Rx.au8_Data[0];
gu8_RegenStick12Pos					:=	RegenStick12_Rx.au8_Data[0];	
	 
(*	 
VDC1_KB_Rx.au8_Data[0];
VDC1_KB_Rx.au8_Data[1];
VDC1_KB_Rx.au8_Data[2];
VDC1_KB_Rx.au8_Data[3];
VDC1_KB_Rx.au8_Data[4];
VDC1_KB_Rx.au8_Data[5];
VDC1_KB_Rx.au8_Data[6];
VDC1_KB_Rx.au8_Data[7];
*)		

gq_Bob_Handbrake_CAN	:=	Bob_Handbrake_Rx.au8_Data[0].0;
gu8_Bob_BrakePos_CAN	:=	Bob_Brake_Rx.au8_Data[1];
	
gu8_Bob_Accel_CAN		:=	Bob_Accel_Rx.au8_Data[1];
gu8_Bob_RegenSelector_CAN	:=	Bob_RegenSelector_Rx.au8_Data[4];
	
IF (Bob_WheelSpeed_Rx.au8_Data[0] <> 254 AND Bob_WheelSpeed_Rx.au8_Data[1] <> 254) THEN
	gu16_Bob_RightDrive_CAN	:=	USINT_TO_UINT(Bob_WheelSpeed_Rx.au8_Data[0]) + SHL(USINT_TO_UINT(Bob_WheelSpeed_Rx.au8_Data[1]), 8);
	hq_Bob_RightDrive_Compromised := FALSE;
ELSE
	IF (hq_Bob_LeftDrive_Compromised = FALSE) THEN
		gu16_Bob_RightDrive_CAN := gu16_Bob_LeftDrive_CAN;
	ELSIF (hq_Bob_RightFront_Compromised = FALSE) THEN
		gu16_Bob_RightDrive_CAN := gu16_Bob_RightFront_CAN;
	ELSIF (hq_Bob_LeftFront_Compromised = FALSE) THEN
		gu16_Bob_RightDrive_CAN := gu16_Bob_LeftFront_CAN;
	ELSE
		gu16_Bob_RightDrive_CAN := 0;
	END_IF
	hq_Bob_RightDrive_Compromised := TRUE;
END_IF
IF (Bob_WheelSpeed_Rx.au8_Data[2] <> 254 AND Bob_WheelSpeed_Rx.au8_Data[3] <> 254) THEN
	gu16_Bob_LeftDrive_CAN	:=	USINT_TO_UINT(Bob_WheelSpeed_Rx.au8_Data[2]) + SHL(USINT_TO_UINT(Bob_WheelSpeed_Rx.au8_Data[3]), 8);
	hq_Bob_LeftDrive_Compromised := FALSE;
ELSE
	IF (hq_Bob_RightDrive_Compromised = FALSE) THEN
		gu16_Bob_LeftDrive_CAN := gu16_Bob_RightDrive_CAN;
	ELSIF (hq_Bob_RightFront_Compromised = FALSE) THEN
		gu16_Bob_LeftDrive_CAN := gu16_Bob_RightFront_CAN;
	ELSIF (hq_Bob_LeftFront_Compromised = FALSE) THEN
		gu16_Bob_LeftDrive_CAN := gu16_Bob_LeftFront_CAN;
	ELSE
		gu16_Bob_LeftDrive_CAN := 0;
	END_IF
	hq_Bob_LeftDrive_Compromised := TRUE;
END_IF
IF (Bob_WheelSpeed_Rx.au8_Data[4] <> 254 AND Bob_WheelSpeed_Rx.au8_Data[5] <> 254) THEN
	gu16_Bob_RightFront_CAN	:=	USINT_TO_UINT(Bob_WheelSpeed_Rx.au8_Data[4]) + SHL(USINT_TO_UINT(Bob_WheelSpeed_Rx.au8_Data[5]), 8);
	hq_Bob_RightFront_Compromised := FALSE;
ELSE
	IF (hq_Bob_RightDrive_Compromised = FALSE) THEN
		gu16_Bob_RightFront_CAN := gu16_Bob_RightDrive_CAN;
	ELSIF (hq_Bob_LeftDrive_Compromised = FALSE) THEN
		gu16_Bob_RightFront_CAN := gu16_Bob_LeftDrive_CAN;
	ELSIF (hq_Bob_LeftFront_Compromised = FALSE) THEN
		gu16_Bob_RightFront_CAN := gu16_Bob_LeftFront_CAN;
	ELSE
		gu16_Bob_RightFront_CAN := 0;
	END_IF
	hq_Bob_RightFront_Compromised := TRUE;
END_IF
IF (Bob_WheelSpeed_Rx.au8_Data[6] <> 254 AND Bob_WheelSpeed_Rx.au8_Data[7] <> 254) THEN
	gu16_Bob_LeftFront_CAN	:=	USINT_TO_UINT(Bob_WheelSpeed_Rx.au8_Data[6]) + SHL(USINT_TO_UINT(Bob_WheelSpeed_Rx.au8_Data[7]), 8);
	hq_Bob_LeftFront_Compromised := FALSE;
ELSE
	IF (hq_Bob_RightDrive_Compromised = FALSE) THEN
		gu16_Bob_LeftFront_CAN := gu16_Bob_RightDrive_CAN;
	ELSIF (hq_Bob_LeftDrive_Compromised = FALSE) THEN
		gu16_Bob_LeftFront_CAN := gu16_Bob_LeftDrive_CAN;
	ELSIF (hq_Bob_RightFront_Compromised = FALSE) THEN
		gu16_Bob_LeftFront_CAN := gu16_Bob_RightFront_CAN;
	ELSE
		gu16_Bob_LeftFront_CAN := 0;
	END_IF
	hq_Bob_LeftFront_Compromised := TRUE;
END_IF
	 
IF (hq_Bob_RightDrive_Compromised = TRUE OR
	hq_Bob_LeftDrive_Compromised = TRUE OR
	hq_Bob_RightFront_Compromised = TRUE OR
	hq_Bob_LeftFront_Compromised = TRUE ) THEN

	gq_Bob_WheelSpeedSensor_Fail := TRUE;
ELSE
	gq_Bob_WheelSpeedSensor_Fail := FALSE;
END_IF

gu8_Bob_ServiceBrakeAirPressCircuit1_CAN	:=	Bob_J1939_AirPressure_Rx.au8_Data[2];
gu8_Bob_ServiceBrakeAirPressCircuit2_CAN	:=	Bob_J1939_AirPressure_Rx.au8_Data[3];
gu8_Bob_AirSuspensionSupplyPress_CAN		:=	Bob_J1939_AirPressure_Rx.au8_Data[5];
gq_Bob_AirCompressorStatus_CAN				:=	Bob_J1939_AirPressure_Rx.au8_Data[6].0;

		 
(*Temperature_Rx.au8_Data[0];*)
	 
IF (gu8_ChassisType = CHASSIS_DENNIS) THEN
	(*gq_StabTracDisable_Rx	:=	Dennis_StabTracDisable_Rx.au8_Data[0].3;*)
	gq_StabTracDisable_Rx	:=	USINT_TO_BOOL(gu8_EBC1_ASROffroadSwitch);
ELSIF (gu8_ChassisType = CHASSIS_BOB OR gu8_ChassisType = CHASSIS_ESTARGLIDER) THEN
	gq_StabTracDisable_Rx	:=	Bob_Brake_Rx.au8_Data[4].2;
END_IF
				  
{endregion}
	 
{region "Comms Loss Check"}
Accelerator_Dennis_Rx_Timer(IN := NOT(Accelerator_Dennis_Rx.q_NewData), PT := T#3S);
Brake_Dennis_Rx_Timer(IN := NOT(EBC1_KB_Rx.q_NewData), PT := T#3S);
GearSelect_Dennis_Rx_Timer(IN := NOT(GearSelect_Dennis_Rx.q_NewData), PT := T#3S);
Airpressure_Dennis_Rx_Timer(IN := NOT(Airpressure_Dennis_Rx.q_NewData), PT := T#3S);
IF (Accelerator_Dennis_Rx_Timer.Q = TRUE AND Brake_Dennis_Rx_Timer.Q = TRUE AND
	GearSelect_Dennis_Rx_Timer.Q = TRUE AND Airpressure_Dennis_Rx_Timer.Q = TRUE) THEN
	gq_Dennis_CAN1_CommsLoss	:=	TRUE;
ELSE
	gq_Dennis_CAN1_CommsLoss	:=	FALSE;
END_IF
{endregion}
	 

gu8_Merc_AirComepressor_Rq	:=	BOOL_TO_USINT(Merc_AIR1_EAPU.au8_Data[6].0) + SHL(BOOL_TO_USINT(Merc_AIR1_EAPU.au8_Data[6].1), 1);
IF ((*gu8_Merc_AirComepressor_Rq*)gq_Bob_AirCompressorStatus_CAN = TRUE(*1*)) THEN
	gq_Merc_AirComp_Rq := TRUE;
ELSE
	gq_Merc_AirComp_Rq := FALSE;
END_IF	
	 
CAN1_RxConversion();

END_PROGRAM

// Application/UserCode/MCU/Dennis_Regen
PROGRAM Dennis_Regen
VAR
	DennisRegen: CTUD;
	RegenCounterValue: WORD := 4;
END_VAR

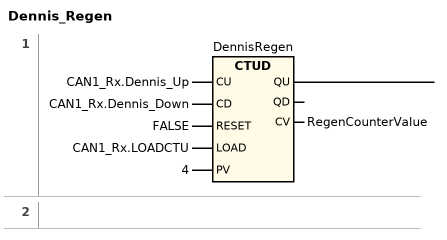
// NETWORK 1
DennisRegen(
    CU := CAN1_Rx.Dennis_Up,
    CD := CAN1_Rx.Dennis_Down,
    RESET := FALSE,
    LOAD := CAN1_Rx.LOADCTU,
    PV := 4,
    CV => RegenCounterValue); // CTUD

// NETWORK 2

END_PROGRAM

// Application/UserCode/CAN1/CAN1_RxConversion
PROGRAM CAN1_RxConversion
VAR
END_VAR
VAR CONSTANT
	NEUTRAL	:	USINT	:=	16#7D;
	DRIVE	:	USINT	:=	16#FC;
	REVERSE	:	USINT	:=	16#DF;
	
	AIRPRESSURE_CF	:	REAL	:=	0.08;
	
	FRONTAXLESPEED_CF	:	REAL	:=	0.00390625;
	RELATIVESPEED_CF	:	REAL	:=	0.0625;
	RELATIVESPEED_OFFSET	:	REAL	:=	-7.8125;
END_VAR


IF  gu8_GearSelector_Dennis_Rx = NEUTRAL AND gq_BrakeSwitch AND gr_VehicleSpeed_kmph <1 AND gr_VehicleSpeed_kmph >-1 THEN
	gq_Neutral_Dennis_Rq	:=	TRUE;
	gq_Drive_Dennis_Rq		:=	FALSE;
	gq_Reverse_Dennis_Rq	:=	FALSE;
ELSIF gu8_GearSelector_Dennis_Rx = DRIVE AND gq_BrakeSwitch AND gr_VehicleSpeed_kmph > -1 THEN
	gq_Neutral_Dennis_Rq	:=	FALSE;
	gq_Drive_Dennis_Rq		:=	TRUE;
	gq_Reverse_Dennis_Rq	:=	FALSE;
ELSIF gu8_GearSelector_Dennis_Rx = REVERSE AND gq_BrakeSwitch AND gr_VehicleSpeed_kmph < 1 THEN
	gq_Neutral_Dennis_Rq	:=	FALSE;
	gq_Drive_Dennis_Rq		:=	FALSE;
	gq_Reverse_Dennis_Rq	:=	TRUE;
ELSE
	;
END_IF
	
IF (gu8_EBC1_ABSActive = 1) THEN
	gq_ABSActive	:=	TRUE;
ELSE
	gq_ABSActive	:=	FALSE;
END_IF

	
gr_EBC2_KB_FrontAxleSpeed				:=	gu16_EBC2_KB_FrontAxleSpeed_Rx * FRONTAXLESPEED_CF;
gr_EBC2_KB_FrontLeftRelSpd				:=	gu16_EBC2_KB_FrontLeftRelSpd_Rx * RELATIVESPEED_CF + RELATIVESPEED_OFFSET;
gr_EBC2_KB_FrontRightRelSpd				:=	gu16_EBC2_KB_FrontRightRelSpd_Rx * RELATIVESPEED_CF + RELATIVESPEED_OFFSET;
gr_EBC2_KB_RearLeft1RelSpd				:=	gu16_EBC2_KB_RearLeft1RelSpd_Rx * RELATIVESPEED_CF + RELATIVESPEED_OFFSET;
gr_EBC2_KB_RearRight1RelSpd				:=	gu16_EBC2_KB_RearRight1RelSpd_Rx * RELATIVESPEED_CF + RELATIVESPEED_OFFSET;
gr_EBC2_KB_RearLeft2RelSpd				:=	gu16_EBC2_KB_RearLeft2RelSpd_Rx * RELATIVESPEED_CF + RELATIVESPEED_OFFSET;
gr_EBC2_KB_RearRight2RelSpd				:=	gu16_EBC2_KB_RearRight2RelSpd_Rx * RELATIVESPEED_CF + RELATIVESPEED_OFFSET;
		

gr_Bob_Accel	:=	(USINT_TO_REAL(gu8_Bob_Accel_CAN) / 250);
IF (gu8_Bob_BrakePos_CAN > 0) THEN
	gq_Bob_Brake_CAN	:=	TRUE;
ELSE
	gq_Bob_Brake_CAN	:=	FALSE;
END_IF

gr_Bob_ServiceBrakeAirPressCircuit1		:=	gu8_Bob_ServiceBrakeAirPressCircuit1_CAN * AIRPRESSURE_CF;
gr_Bob_ServiceBrakeAirPressCircuit2		:=	gu8_Bob_ServiceBrakeAirPressCircuit2_CAN * AIRPRESSURE_CF;
gr_Bob_AirSuspensionSupplyPress			:=	gu8_Bob_AirSuspensionSupplyPress_CAN * AIRPRESSURE_CF;

END_PROGRAM

// Application/UserCode/CAN Function Blocks/CAN1/Receive_CAN1_EXD_28bit
FUNCTION_BLOCK Receive_CAN1_EXD_28bit
VAR_INPUT
	u32_COBID	:	DWORD;
END_VAR
VAR_OUTPUT
	q_NewData	:	BOOL;
	au8_Data	:	ARRAY [0..7] OF BYTE;
	u8_Length	:	BYTE;
END_VAR
VAR
	hq_Initialise	:	BOOL	:=	FALSE;
	ht_RxMessage	:	t_CANReceive;
	ht_MsgRx		:	Callback_Receive_CAN1;
END_VAR



IF (hq_Initialise = FALSE) THEN
	(*
	(*11 bit*)
	G_CAN1_Channel.AddCOBID(i_CobId := u32_COBID,
							i_itfCallback := ht_RxMessage,
							i_Argument := ADR(ht_RxMessage));
	*)
	(*29 bit*)
	G_CAN1_Channel.AddCOBID(i_CobId := u32_COBID OR EPEC_CANVXD.MASK_29BIT,
							i_itfCallback := ht_MsgRx,
							i_Argument := ADR(ht_RxMessage));
	G_CAN1_Channel.SetMask(i_CobID := u32_COBID OR EPEC_CANVXD.MASK_29BIT, i_Mask := 16#0CFF0211 OR 16#0C010305 (*OR EPEC_CANVXD.MASK_29BIT*));

	hq_Initialise	:=	TRUE;
END_IF


IF (ht_RxMessage.q_NewDataRxed = TRUE) THEN
	au8_Data	:=	ht_RxMessage.Data;
	u8_Length	:=	ht_RxMessage.Len;
	q_NewData	:=	TRUE;
	ht_RxMessage.q_NewDataRxed	:=	FALSE;
ELSE
	q_NewData	:=	FALSE;
END_IF

END_FUNCTION_BLOCK

// Application/UserCode/CAN3/CAN3_Rx
PROGRAM CAN3_Rx
VAR
	GearSelect_Bob_Rx	:	Receive_CAN3_EXD_28bit;
	MercStalk_Rx		:	Receive_CAN3_EXD;
	Merc_AIR1_EAPU: Receive_CAN3_EXD;
	Mode_Button: BOOL;
	Up_Button: BOOL;
	Down_Button: BOOL;
END_VAR


GearSelect_Bob_Rx	(u32_COBID	:=	16#0C010305,
						q_NewData => ,
						au8_Data => ,
						u8_Length => 			);
						
MercStalk_Rx	(u32_COBID	:=	16#18FF0400,
						q_NewData => ,
						au8_Data => ,
						u8_Length => 			);
(*COPIED FROM CAN 1*)					
Merc_AIR1_EAPU	(u32_COBID := 16#14FEAE30,
		 	q_NewData => ,
			au8_Data => ,
			u8_Length =>			);	
			
IF GearSelect_Bob_Rx.au8_Data[5] = 16#7F THEN
	Mode_Button := TRUE;
ELSE
	Mode_Button := FALSE;
	END_IF

IF GearSelect_Bob_Rx.au8_Data[2] = 16#F9 THEN
	Up_Button := TRUE;
ELSE
	Up_Button := FALSE;
	END_IF

IF GearSelect_Bob_Rx.au8_Data[2] = 16#F7 THEN
	Down_Button := TRUE;
ELSE
	Down_Button := FALSE;
	END_IF
	
(*gu8_Merc_AirComepressor_Rq	:=	BOOL_TO_USINT(Merc_AIR1_EAPU.au8_Data[6].0) + SHL(BOOL_TO_USINT(Merc_AIR1_EAPU.au8_Data[6].1), 1);
IF (gu8_Merc_AirComepressor_Rq = 1) THEN 
	gq_Merc_AirComp_Rq := TRUE;
ELSE
	gq_Merc_AirComp_Rq := FALSE;
END_IF*)

(******)					
gu8_GearSelector_Bob_Rx	:=	GearSelect_Bob_Rx.au8_Data[2];

gu8_Merc_AutoManualSwitch	:=	BOOL_TO_USINT(MercStalk_Rx.au8_Data[0].0) + SHL(BOOL_TO_USINT(MercStalk_Rx.au8_Data[0].1), 1);
(*MercStalk_Rx.au8_Data[0];
MercStalk_Rx.au8_Data[1];*)
gu8_Merc_GearSelectSwitch	:=	BOOL_TO_USINT(MercStalk_Rx.au8_Data[2].2) + SHL(BOOL_TO_USINT(MercStalk_Rx.au8_Data[2].3), 1) +
								SHL(BOOL_TO_USINT(MercStalk_Rx.au8_Data[2].4), 2) + SHL(BOOL_TO_USINT(MercStalk_Rx.au8_Data[2].5), 3);
(*MercStalk_Rx.au8_Data[2];
MercStalk_Rx.au8_Data[3];*)
gq_Merc_Neutral				:=	MercStalk_Rx.au8_Data[4].0;
gq_Merc_Drive				:=	MercStalk_Rx.au8_Data[4].1;
gq_Merc_Reverse				:=	MercStalk_Rx.au8_Data[4].2;
(*MercStalk_Rx.au8_Data[4];
MercStalk_Rx.au8_Data[5];
MercStalk_Rx.au8_Data[6];
MercStalk_Rx.au8_Data[7];*)

CAN3_RxConversion();

END_PROGRAM

// Application/UserCode/CAN3/CAN3_RxConversion
PROGRAM CAN3_RxConversion
VAR
	;
END_VAR
VAR CONSTANT
	NEUTRAL	:	USINT	:=	16#7D;
	DRIVE	:	USINT	:=	16#FC;
	REVERSE	:	USINT	:=	16#DF;
	NOPRESS	:	USINT	:=	16#7C;
END_VAR



IF (gu8_GearSelector_Bob_Rx = NEUTRAL) AND (gu8_GearSelector_Bob_Rx <> 224) AND gq_BrakeSwitch = TRUE AND gr_VehicleSpeed_kmph <0.001 AND gr_VehicleSpeed_kmph >-0.001 THEN
	gq_Neutral_Bob_Rq	:=	TRUE;
	gq_Drive_Bob_Rq		:=	FALSE;
	gq_Reverse_Bob_Rq	:=	FALSE;
ELSIF (gu8_GearSelector_Bob_Rx = DRIVE) AND (gu8_GearSelector_Bob_Rx <> 224) AND gq_BrakeSwitch = TRUE AND gr_VehicleSpeed_kmph > -0.001 THEN
	gq_Neutral_Bob_Rq	:=	FALSE;
	gq_Drive_Bob_Rq		:=	TRUE;
	gq_Reverse_Bob_Rq	:=	FALSE;
ELSIF (gu8_GearSelector_Bob_Rx = REVERSE) AND (gu8_GearSelector_Bob_Rx <> 224) AND gq_BrakeSwitch = TRUE AND gr_VehicleSpeed_kmph < 0.001 THEN
	gq_Neutral_Bob_Rq	:=	FALSE;
	gq_Drive_Bob_Rq		:=	FALSE;
	gq_Reverse_Bob_Rq	:=	TRUE;
ELSE
	;
END_IF

END_PROGRAM

// Application/UserCode/CAN Function Blocks/CAN3/Receive_CAN3_EXD_28bit
FUNCTION_BLOCK Receive_CAN3_EXD_28bit
VAR_INPUT
	u32_COBID	:	DWORD;
END_VAR
VAR_OUTPUT
	q_NewData	:	BOOL;
	au8_Data	:	ARRAY [0..7] OF BYTE;
	u8_Length	:	BYTE;
END_VAR
VAR
	hq_Initialise	:	BOOL	:=	FALSE;
	ht_RxMessage	:	t_CANReceive;
	ht_MsgRx		:	Callback_Receive_CAN1;
END_VAR



IF (hq_Initialise = FALSE) THEN
	(*
	IF (u32_COBID > 16#7FF) THEN
		(*29 bit*)
		;
	ELSE
		(*11 bit*)
		;
	END_IF
	*)
	(*
	(*11 bit*)
	G_CAN3_Channel.AddCOBID(i_CobId := u32_COBID,
							i_itfCallback := ht_RxMessage,
							i_Argument := ADR(ht_RxMessage));
	*)
	(*29 bit*)
	G_CAN3_Channel.AddCOBID(i_CobId := u32_COBID OR EPEC_CANVXD.MASK_29BIT,
							i_itfCallback := ht_MsgRx,
							i_Argument := ADR(ht_RxMessage));
	G_CAN3_Channel.SetMask(i_CobID := u32_COBID OR EPEC_CANVXD.MASK_29BIT, i_Mask := 16#0C010305);

	hq_Initialise	:=	TRUE;
END_IF


IF (ht_RxMessage.q_NewDataRxed = TRUE) THEN
	au8_Data	:=	ht_RxMessage.Data;
	u8_Length	:=	ht_RxMessage.Len;
	q_NewData	:=	TRUE;
	ht_RxMessage.q_NewDataRxed	:=	FALSE;
ELSE
	q_NewData	:=	FALSE;
END_IF

END_FUNCTION_BLOCK

// Application/UserCode/CAN Function Blocks/CAN3/Receive_CAN3_EXD
FUNCTION_BLOCK Receive_CAN3_EXD
VAR_INPUT
	u32_COBID	:	DWORD;
END_VAR
VAR_OUTPUT
	q_NewData	:	BOOL;
	au8_Data	:	ARRAY [0..7] OF BYTE;
	u8_Length	:	BYTE;
END_VAR
VAR
	hq_Initialise	:	BOOL	:=	FALSE;
	ht_RxMessage	:	t_CANReceive;
	ht_MsgRx		:	Callback_Receive_CAN1;
END_VAR



IF (hq_Initialise = FALSE) THEN
	(*
	IF (u32_COBID > 16#7FF) THEN
		(*29 bit*)
		;
	ELSE
		(*11 bit*)
		;
	END_IF
	*)
	(*
	(*11 bit*)
	G_CAN3_Channel.AddCOBID(i_CobId := u32_COBID,
							i_itfCallback := ht_RxMessage,
							i_Argument := ADR(ht_RxMessage));
	*)
	(*29 bit*)
	G_CAN3_Channel.AddCOBID(i_CobId := u32_COBID OR EPEC_CANVXD.MASK_29BIT,
							i_itfCallback := ht_MsgRx,
							i_Argument := ADR(ht_RxMessage));
	G_CAN3_Channel.SetMask(i_CobID := u32_COBID OR EPEC_CANVXD.MASK_29BIT, (*i_Mask := 16#0C009000 OR*) EPEC_CANVXD.MASK_29BIT);

	hq_Initialise	:=	TRUE;
END_IF


IF (ht_RxMessage.q_NewDataRxed = TRUE) THEN
	au8_Data	:=	ht_RxMessage.Data;
	u8_Length	:=	ht_RxMessage.Len;
	q_NewData	:=	TRUE;
	ht_RxMessage.q_NewDataRxed	:=	FALSE;
ELSE
	q_NewData	:=	FALSE;
END_IF

END_FUNCTION_BLOCK

// Application/UserCode/CAN4/CAN4_Rx
PROGRAM CAN4_Rx
VAR
	Handbrake_Rx	:	Receive_CAN4_EXD;
	Handbrake_Rx_Timer	:	TON;
	
	
	
	
	
	
END_VAR

Handbrake_Rx(u32_COBID	:=	16#18FEF1F2,
			q_NewData => ,
			au8_Data => ,
			u8_Length => 			);
			
				
gq_Handbrake_CAN	:=	Handbrake_Rx.au8_Data[0].2;				
				
Handbrake_Rx_Timer(IN := NOT(Handbrake_Rx.q_NewData), PT := t#10s);

END_PROGRAM

// Application/UserCode/ePTO/EPTO_Rx
PROGRAM EPTO_Rx
VAR
	ePTO_Rx			:	Receive_CAN4_STD;
	ePTO_Dennis_Rx	:	Receive_CAN4_EXD;
	SkaiUnit_Temp_Rx	:	Receive_CAN4_STD;
END_VAR


ePTO_Rx		(u32_COBID	:=	16#141,
						q_NewData => ,
						au8_Data => ,
						u8_Length => 		);
						
ePTO_Dennis_Rx (u32_COBID	:=	16#2CFF1355,
						q_NewData => ,
						au8_Data => ,
						u8_Length => 		);
						
SkaiUnit_Temp_Rx (u32_COBID	:=	16#1BA,
						q_NewData => ,
						au8_Data => ,
						u8_Length => 		);

IF (gu8_ChassisType = CHASSIS_DENNIS) THEN
	gu8_ePTO_ActivationByte	:=	ePTO_Dennis_Rx.au8_Data[3]; (*4*)
ELSE
	gu8_ePTO_ActivationByte	:=	ePTO_Rx.au8_Data[4];				
END_IF					

gs16_InverterTemp	:= SkaiUnit_Temp_Rx.au8_Data[0] - 40;
gs16_MotorTemp		:= SkaiUnit_Temp_Rx.au8_Data[1] - 40; (*Use this for the ePTO activation instead of the boolean trigger*)

END_PROGRAM

// Application/UserCode/Main Program/Chassis_Parameters
PROGRAM Chassis_Parameters
VAR
	har_AccelInput	:	ARRAY [0..10] OF REAL;
	hu8_InputCounter	:	USINT;
	hr_SumAccelPedal		:	REAL;
	hr_AverageAccelPedal	:	REAL;
	hu8_Counter	:	USINT;
	
	hr_AccelAveraging : ARRAY [0..9] OF REAL;
	CycleCounter	:	USINT	:=	0;
	Sum_Counter		:	USINT	:=	0;
	hr_AccelSum		:	REAL	:=	0;
END_VAR
VAR CONSTANT
	(*MCU*)
	OPERATIONAL		:	USINT	:=	4;
	(*Iveco*)
	MAX_THROTTLE	:	UINT	:=	6000;
	THROTTLE_OFFSET	:	UINT	:=	750;
	(*Dennis*)
	MAX_THROTTLE_CAN	:	USINT	:=	250;
	
	AIRPRESSURE_CF	:	REAL	:=	0.08;
	
	(*Air Compressor Limits*)
	LOWAIRPRESSURE_DENNIS : REAL := 8.0;
END_VAR
VAR
	HIGHAIRPRESSURE_DENNIS : REAL := 10.3; //10.5
END_VAR
VAR CONSTANT
	LOWAIRPRESSURE_BOB : REAL := 9.8;
	HIGHAIRPRESSURE_BOB : REAL := 11.9;
	LOWAIRPRESSURE_IVECO : REAL := 8.2;
	HIGHAIRPRESSURE_IVECO : REAL := 10;
	LOWAIRPRESSURE_GLIDER : REAL := 9.8;
	
	
	HIGHAIRPRESSURE_GLIDER : REAL := 11.9;
END_VAR


CASE gu8_ChassisType OF
	CHASSIS_DENNIS:
		gq_HandBrake			:=	gq_Handbrake_CAN;
		gq_BrakeSwitch			:=	USINT_TO_BOOL(gu8_EBC1_EBSBrakeSwitch);
		gu8_BrakePedal_Perc		:=	gu8_EBC1_BrakePedalPosition; (*Value given in same message as the switch active*)
		IF (gu8_AccelPedal_Dennis_Rx <= MAX_THROTTLE_CAN) THEN
			(*hr_AccelAveraging[CycleCounter]*)gr_AccelPedal_Perc	:=	(USINT_TO_REAL(gu8_AccelPedal_Dennis_Rx) / MAX_THROTTLE_CAN);	
		ELSE
			(*hr_AccelAveraging[CycleCounter]*)gr_AccelPedal_Perc		:=	0;
		END_IF
		(*IF (gq_Dennis_Accel_NewData = TRUE) THEN
			CycleCounter := CycleCounter + 1;
		END_IF
		IF (CycleCounter > 9) THEN
			CycleCounter := 0;
		END_IF
		hr_AccelSum	:=	0;
		FOR Sum_Counter := 0 TO 9 DO
			hr_AccelSum	:=	hr_AccelSum + hr_AccelAveraging[Sum_Counter];
		END_FOR
		gr_AccelPedal_Perc		:=	hr_AccelSum / 10;*)
		
		gq_Gear_Neutral_Rq		:=	gq_Neutral_Dennis_Rq;
		gq_Gear_Drive_Rq		:=	gq_Drive_Dennis_Rq;
		gq_Gear_Reverse_Rq		:=	gq_Reverse_Dennis_Rq;
		
		gr_J1939_AirSuspensionSupplyPress		:=	USINT_TO_REAL(gu8_Dennis_AirPressureSusp_Rx) * AIRPRESSURE_CF;
		gr_J1939_ServiceBrakeAirPressCircuit1	:=	USINT_TO_REAL(gu8_Dennis_AirPressureBrake1_Rx) * AIRPRESSURE_CF;
		gr_J1939_ServiceBrakeAirPressCircuit2	:=	USINT_TO_REAL(gu8_Dennis_AirPressureBrake2_Rx) * AIRPRESSURE_CF;
		
		gu8_RegenSelector		:=	1; (*Put the same as whatever the Iveco would receive for position 2*)
		
		gr_LowAirPressure_Intro		:=	LOWAIRPRESSURE_DENNIS;
		gr_HighAirPressure_CutOff	:=	HIGHAIRPRESSURE_DENNIS;
		
	CHASSIS_BOB:
		gq_HandBrake			:=	gq_Bob_Handbrake_CAN;
		gq_BrakeSwitch			:=	gq_Bob_Brake_CAN;
		gu8_BrakePedal_Perc		:=	REAL_TO_USINT(gu8_Bob_BrakePos_CAN / 250) * 100; (*Not used currently*)
		gr_AccelPedal_Perc		:=	gr_Bob_Accel;
		gq_Gear_Neutral_Rq		:=	gq_Neutral_Bob_Rq;
		gq_Gear_Drive_Rq		:=	gq_Drive_Bob_Rq;
		gq_Gear_Reverse_Rq		:=	gq_Reverse_Bob_Rq;
		
		(*IF (gu8_RegenStick01Pos = 16#CF) THEN
			gu8_RegenSelector	:=	0; (*Find out wtf the selector is and put it here same for Daimler*)
		ELSIF (gu8_RegenStick01Pos = 16#DF) THEN
			IF (gu8_RegenStick12Pos = 16#DE) THEN
				gu8_RegenSelector	:=	1;
			ELSIF (gu8_RegenStick12Pos = 16#FC) THEN
				gu8_RegenSelector	:=	2;
			END_IF
		END_IF*)
		gu8_RegenSelector	:=	gu8_Bob_RegenSelector_CAN;
		(*Needs to be new SA*)
		gr_J1939_AirSuspensionSupplyPress		:=	gr_Bob_AirSuspensionSupplyPress;
		gr_J1939_ServiceBrakeAirPressCircuit1	:=	gr_Bob_ServiceBrakeAirPressCircuit1;
		gr_J1939_ServiceBrakeAirPressCircuit2	:=	gr_Bob_ServiceBrakeAirPressCircuit2;
		
		gr_LowAirPressure_Intro		:=	LOWAIRPRESSURE_BOB;
		gr_HighAirPressure_CutOff	:=	HIGHAIRPRESSURE_BOB;
		
	CHASSIS_IVECO:
		gq_HandBrake			:=	BYTE_TO_BOOL(J1939_CAN1.In.CCVS.CCVS_ParkingBrakeSwitch);
		gq_BrakeSwitch			:=	BYTE_TO_BOOL(J1939_CAN1.In.CCVS.CCVS_BrakeSwitch);
		gu8_BrakePedal_Perc		:=	0; (*Can't find on the Iveco*)
		
		(*
		har_AccelInput[hu8_InputCounter]	:=	AI_u16_VehicleThrottlePedal1_AI;
		IF (hu8_InputCounter < 10) THEN
			hu8_InputCounter	:=	hu8_InputCounter + 1;
		ELSE
			hu8_InputCounter	:=	0;
		END_IF
		hr_SumAccelPedal	:=	0;
		FOR hu8_Counter := 0 TO 10 DO
			hr_SumAccelPedal	:=	hr_SumAccelPedal + har_AccelInput[hu8_Counter];
		END_FOR
		hr_AverageAccelPedal	:=	hr_SumAccelPedal / 11;*)
		
		IF (AI_u16_VehicleThrottlePedal1_AI > THROTTLE_OFFSET AND gu8_MCU_State = OPERATIONAL) THEN
			gr_AccelPedal_Perc	:=	(UINT_TO_REAL(AI_u16_VehicleThrottlePedal1_AI) - THROTTLE_OFFSET) / (MAX_THROTTLE - THROTTLE_OFFSET);
		ELSE
			gr_AccelPedal_Perc	:=	0;
		END_IF
		(*Do an array of received values then either use a filter or do averaging on the array. New value each program cycle.*)
		
		gq_Gear_Neutral_Rq		:=	DI_q_DirectionSwitch_Neutral_DI;
		gq_Gear_Drive_Rq		:=	DI_q_DirectionSwitch_Drive_DI;
		gq_Gear_Reverse_Rq		:=	DI_q_DirectionSwitch_Reverse_DI;
	
		IF (gu8_RegenStick01Pos = 16#CF) THEN
			gu8_RegenSelector	:=	0;
		ELSIF (gu8_RegenStick01Pos = 16#DF) THEN
			IF (gu8_RegenStick12Pos = 16#DE) THEN
				gu8_RegenSelector	:=	1;
			ELSIF (gu8_RegenStick12Pos = 16#FC) THEN
				gu8_RegenSelector	:=	2;
			END_IF
		END_IF
		
		gr_J1939_AirSuspensionSupplyPress		:=	BYTE_TO_REAL(J1939_CAN1.In.BodyCont.AIR1_AirSuspensionSupplyPress) * AIRPRESSURE_CF;
		gr_J1939_ServiceBrakeAirPressCircuit1	:=	BYTE_TO_REAL(J1939_CAN1.In.BodyCont.AIR1_ServiceBrakeAirPressCircuit1) * AIRPRESSURE_CF;
		gr_J1939_ServiceBrakeAirPressCircuit2	:=	BYTE_TO_REAL(J1939_CAN1.In.BodyCont.AIR1_ServiceBrakeAirPressCircuit2) * AIRPRESSURE_CF;
		(*Charge mode enable / charger detected*)
		(**)
		gr_LowAirPressure_Intro		:=	LOWAIRPRESSURE_IVECO;
		gr_HighAirPressure_CutOff	:=	HIGHAIRPRESSURE_IVECO;
		;

	CHASSIS_ESTARGLIDER:
		gq_HandBrake			:=	gq_Bob_Handbrake_CAN;
		gq_BrakeSwitch			:=	gq_Bob_Brake_CAN;
		gu8_BrakePedal_Perc		:=	REAL_TO_USINT(gu8_Bob_BrakePos_CAN / 250) * 100; (*Not used currently*)
		gr_AccelPedal_Perc		:=	gr_Bob_Accel;
		
		IF (gq_Daimler_PowerShift_Installed = TRUE) THEN
			gq_Gear_Neutral_Rq		:=	gq_Merc_Neutral;
			gq_Gear_Drive_Rq		:=	gq_Merc_Drive;
			gq_Gear_Reverse_Rq		:=	gq_Merc_Reverse;
		ELSE
			gq_Gear_Neutral_Rq		:=	gq_Neutral_Bob_Rq;
			gq_Gear_Drive_Rq		:=	gq_Drive_Bob_Rq;
			gq_Gear_Reverse_Rq		:=	gq_Reverse_Bob_Rq;
		END_IF
		
IF (gq_Daimler_PowerShift_Installed = TRUE AND gq_CAN1_Merc_Gears = TRUE) THEN
			gq_Gear_Neutral_Rq		:=	CAN1_Rx.MercStalk_Rx.au8_Data[4].0;
			gq_Gear_Drive_Rq		:=	CAN1_Rx.MercStalk_Rx.au8_Data[4].1;
			gq_Gear_Reverse_Rq		:=	CAN1_Rx.MercStalk_Rx.au8_Data[4].2;
		ELSE
			gq_Gear_Neutral_Rq		:=	gq_Neutral_Bob_Rq;
			gq_Gear_Drive_Rq		:=	gq_Drive_Bob_Rq;
			gq_Gear_Reverse_Rq		:=	gq_Reverse_Bob_Rq;
		END_IF
		
		gu8_RegenSelector	:=	gu8_Bob_RegenSelector_CAN;
		(*Needs to be new SA*)
		gr_J1939_AirSuspensionSupplyPress		:=	gr_Bob_AirSuspensionSupplyPress;
		gr_J1939_ServiceBrakeAirPressCircuit1	:=	gr_Bob_ServiceBrakeAirPressCircuit1;
		gr_J1939_ServiceBrakeAirPressCircuit2	:=	gr_Bob_ServiceBrakeAirPressCircuit2;
		
		gr_LowAirPressure_Intro		:=	LOWAIRPRESSURE_GLIDER;
		gr_HighAirPressure_CutOff	:=	HIGHAIRPRESSURE_GLIDER;
		
END_CASE


gs16_MaxTemp_degC	:=	MAX(MAX(gs16_Sevcon1_MotorTemp, gs16_Sevcon2_MotorTemp), REAL_TO_INT(gr_MCU_ThermalIndicator));

END_PROGRAM

// Application/UserCode/Cooling Fan/Cooling_Fan
PROGRAM Cooling_Fan
VAR
	Fan_Switch: BOOL := FALSE;
	MCU_Temp_Setpoint: INT := 40;
	Compressor_Temp_Setpoint: INT := 130;
	Comp_Motor_Temp_Setpoint: INT := 85;
	Brusa_1_Cooling_Request_Setpoint: INT := 100; 
	Brusa_2_Cooling_Request_Setpoint: INT := 100; 
	MCU_Temp_Setpoint_OFF: INT := 38;
	Compressor_Temp_Setpoint1: INT := 100;
	Comp_Motor_Temp_Setpoint1: INT := 80;
	Brusa_1_Cooling_Request_Setpoint1: INT := 85; 
	Brusa_2_Cooling_Request_Setpoint1: INT := 85; 
END_VAR

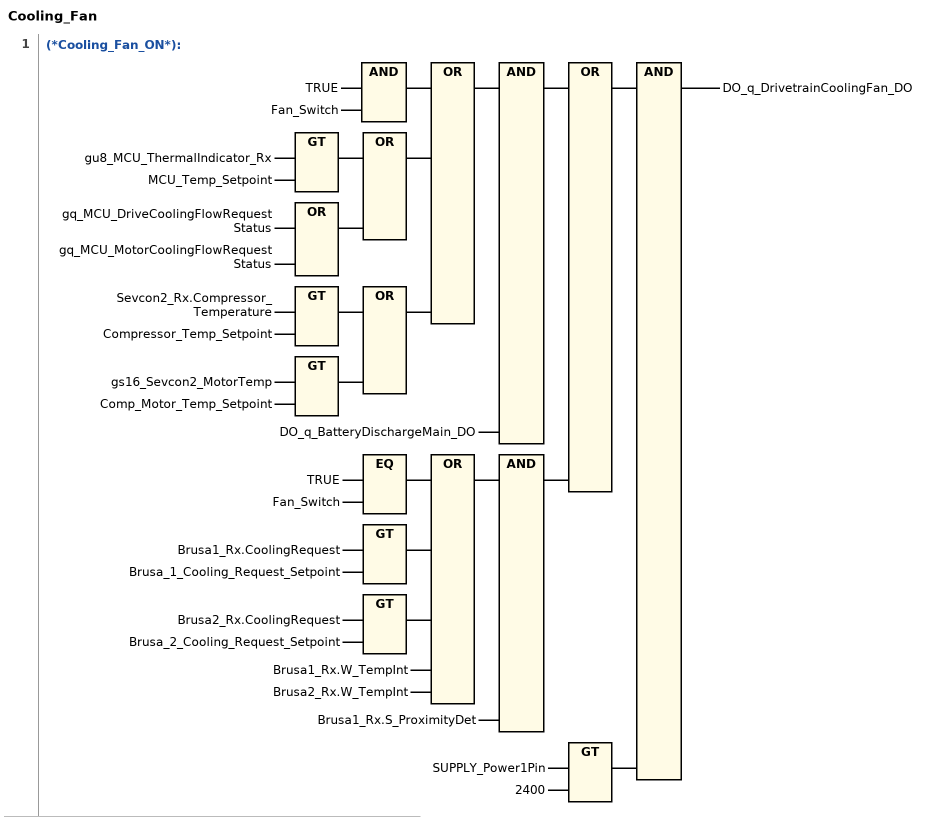
// NETWORK 1
// label: (*Cooling_Fan_ON*)
DO_q_DrivetrainCoolingFan_DO := ((TRUE AND Fan_Switch OR (gu8_MCU_ThermalIndicator_Rx > MCU_Temp_Setpoint OR (gq_MCU_DriveCoolingFlowRequestStatus OR gq_MCU_MotorCoolingFlowRequestStatus)) OR (Sevcon2_Rx.Compressor_Temperature > Compressor_Temp_Setpoint OR gs16_Sevcon2_MotorTemp > Comp_Motor_Temp_Setpoint)) AND DO_q_BatteryDischargeMain_DO OR (TRUE = Fan_Switch OR Brusa1_Rx.CoolingRequest > Brusa_1_Cooling_Request_Setpoint OR Brusa2_Rx.CoolingRequest > Brusa_2_Cooling_Request_Setpoint OR Brusa1_Rx.W_TempInt OR Brusa2_Rx.W_TempInt) AND Brusa1_Rx.S_ProximityDet) AND SUPPLY_Power1Pin > 2400;

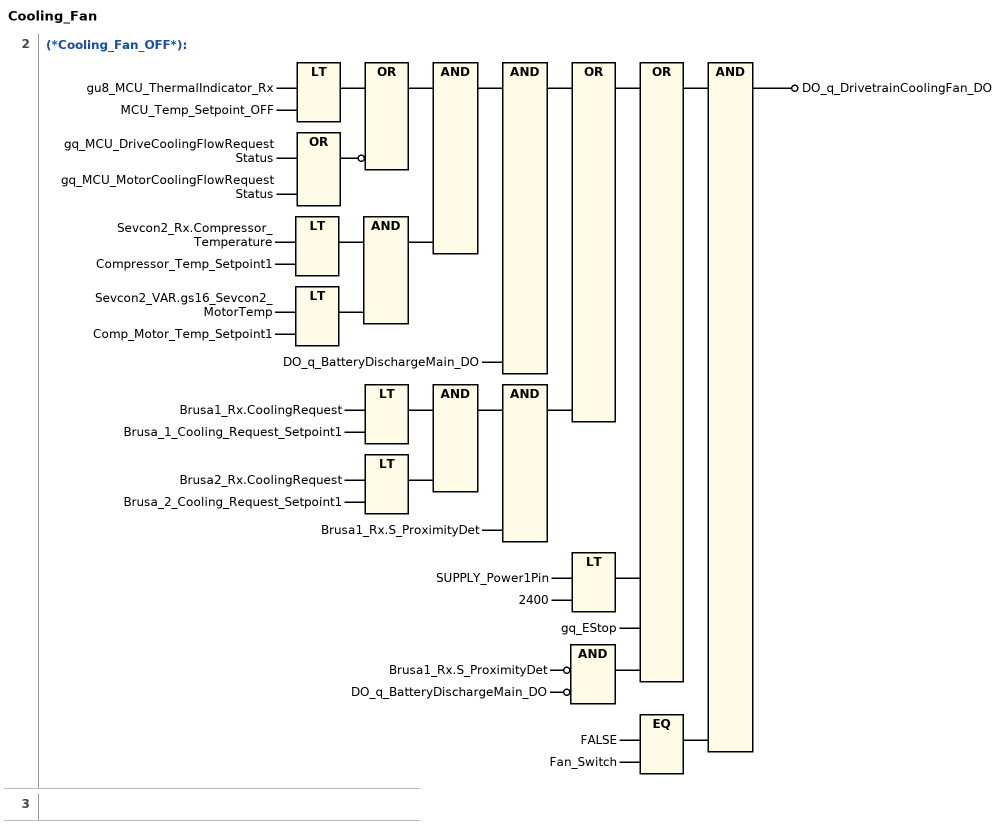
// NETWORK 2
// label: (*Cooling_Fan_OFF*)
DO_q_DrivetrainCoolingFan_DO := NOT (((((gu8_MCU_ThermalIndicator_Rx < MCU_Temp_Setpoint_OFF OR NOT (gq_MCU_DriveCoolingFlowRequestStatus OR gq_MCU_MotorCoolingFlowRequestStatus)) AND (Sevcon2_Rx.Compressor_Temperature < Compressor_Temp_Setpoint1 AND Sevcon2_VAR.gs16_Sevcon2_MotorTemp < Comp_Motor_Temp_Setpoint1)) AND DO_q_BatteryDischargeMain_DO OR (Brusa1_Rx.CoolingRequest < Brusa_1_Cooling_Request_Setpoint1 AND Brusa2_Rx.CoolingRequest < Brusa_2_Cooling_Request_Setpoint1) AND Brusa1_Rx.S_ProximityDet) OR SUPPLY_Power1Pin < 2400 OR gq_EStop OR NOT Brusa1_Rx.S_ProximityDet AND NOT DO_q_BatteryDischargeMain_DO) AND FALSE = Fan_Switch);

// NETWORK 3

END_PROGRAM

// Application/UserCode/Fault Handler/FaultDetection
PROGRAM FaultDetection
VAR
	hq_Dennis_CommsErr	:	BOOL;
	hton_MCU_CutOff_Timer	:	TON;
	hton_DriveMode_CutOff_Timer	:	TON;
	hton_LowCVRecovery_Timer	:	TON;
END_VAR
VAR CONSTANT
	FAULTOFF_STAT	:	USINT	:=	13;
	LV_LOW			:	USINT	:=	22;
END_VAR


IF (gu8_BMSType = BMS_ORION) THEN
	(*BMS1*)
	IF((*DTC1 Flags*)
		OrionBMS1_DTCFlag1_0A07_DischargeLimitEnforcementFault1= TRUE OR
		OrionBMS1_DTCFlag1_0A08_ChargerSafetyRelayFault1= TRUE OR
		OrionBMS1_DTCFlag1_0A09_InternalHardwareFault1= TRUE OR
		OrionBMS1_DTCFlag1_0A0A_InternalHeatskinkThermistorFault= TRUE OR
		OrionBMS1_DTCFlag1_0A0B_InternalSoftwareFault1= TRUE OR
		OrionBMS1_DTCFlag1_0A0C_HighestCellVoltageTooHighFault1= TRUE OR 
		OrionBMS1_DTCFlag1_0A0E_LowestCellVoltageTooLowFault= TRUE OR	
		OrionBMS1_DTCFlag1_0A10_PackTooHotFault1= TRUE OR	
		(*DTC2 Flags*)
		OrionBMS1_DTCFlags2_0A1F_InternalCommunicationFault	OR	
		(*OrionBMS1_DTCFlags2_0A12_CellBalancingStruckOffFault= TRUE OR*)	
		(*OrionBMS1_DTCFlags2_0A80_WeakCellFault= TRUE OR*)
		OrionBMS1_DTCFlags2_0AFA_LowCellVoltageFault= TRUE OR			
		OrionBMS1_DTCFlags2_0A04_OpenWiringFault= TRUE OR
		OrionBMS1_DTCFlags2_0AC0_CurrentSensorFault= TRUE OR				
		OrionBMS1_DTCFlags2_0A0D_HighestCellVoltageOver5vFault= TRUE OR		
		OrionBMS1_DTCFlags2_0A0F_CellASICFault= TRUE OR
		OrionBMS1_DTCFlags2_0A02_WeakPackFault= TRUE OR				
		(*OrionBMS1_DTCFlags2_0A81_FanMonitorFault= TRUE OR*)				
		(*OrionBMS1_DTCFlags2_0A9C_ThermistorFault= TRUE OR*)			
		OrionBMS1_DTCFlags2_0100_ExternalCommunicationFault= TRUE OR		
		OrionBMS1_DTCFlags2_0560_RedundantPowerSupplyFault= TRUE OR	
		OrionBMS1_DTCFlags2_0AA6_HighVoltageIsolatonFault= TRUE OR
		OrionBMS1_DTCFlags2_0A05_InputPowerSupplyFault= TRUE OR	
		OrionBMS1_DTCFlags2_0A06_ChargeLimitEnforcementFault= TRUE OR
		gq_OrionBMS1_CommsLoss = TRUE) THEN
			gq_BMS1_Orion_Error	:=	TRUE;
	ELSE
			gq_BMS1_Orion_Error	:=	FALSE;
	END_IF
	(*BMS2*)
	IF((*DTC1 Flags*)
		OrionBMS2_DTCFlag1_0A07_DischargeLimitEnforcementFault1= TRUE OR
		OrionBMS2_DTCFlag1_0A08_ChargerSafetyRelayFault1= TRUE OR
		OrionBMS2_DTCFlag1_0A09_InternalHardwareFault1= TRUE OR
		OrionBMS2_DTCFlag1_0A0A_InternalHeatskinkThermistorFault= TRUE OR
		OrionBMS2_DTCFlag1_0A0B_InternalSoftwareFault1= TRUE OR
		OrionBMS2_DTCFlag1_0A0C_HighestCellVoltageTooHighFault1= TRUE OR 
		OrionBMS2_DTCFlag1_0A0E_LowestCellVoltageTooLowFault= TRUE OR	
		OrionBMS2_DTCFlag1_0A10_PackTooHotFault1= TRUE OR	
		(*DTC2 Flags*)
		OrionBMS2_DTCFlags2_0A1F_InternalCommunicationFault	OR	
		(*OrionBMS2_DTCFlags2_0A12_CellBalancingStruckOffFault= TRUE OR	*)
		(*OrionBMS2_DTCFlags2_0A80_WeakCellFault= TRUE OR*)
		OrionBMS2_DTCFlags2_0AFA_LowCellVoltageFault= TRUE OR			
		OrionBMS2_DTCFlags2_0A04_OpenWiringFault= TRUE OR
		OrionBMS2_DTCFlags2_0AC0_CurrentSensorFault= TRUE OR				
		OrionBMS2_DTCFlags2_0A0D_HighestCellVoltageOver5vFault= TRUE OR		
		OrionBMS2_DTCFlags2_0A0F_CellASICFault= TRUE OR
		OrionBMS2_DTCFlags2_0A02_WeakPackFault= TRUE OR				
		(*OrionBMS2_DTCFlags2_0A81_FanMonitorFault= TRUE OR*)				
		(*OrionBMS2_DTCFlags2_0A9C_ThermistorFault= TRUE OR*)			
		OrionBMS2_DTCFlags2_0100_ExternalCommunicationFault= TRUE OR		
		OrionBMS2_DTCFlags2_0560_RedundantPowerSupplyFault= TRUE OR	
		OrionBMS2_DTCFlags2_0AA6_HighVoltageIsolatonFault= TRUE OR
		OrionBMS2_DTCFlags2_0A05_InputPowerSupplyFault= TRUE OR	
		OrionBMS2_DTCFlags2_0A06_ChargeLimitEnforcementFault= TRUE OR
		gq_OrionBMS2_CommsLoss = TRUE) THEN
			gq_BMS2_Orion_Error	:=	TRUE;
	ELSE
			gq_BMS2_Orion_Error	:=	FALSE;
	END_IF
END_IF
	 
IF gq_BMS1_Orion_Error = TRUE THEN
	gq_BMS1_Error	:=	TRUE;
ELSE
	gq_BMS1_Error	:=	FALSE;		 
END_IF
IF gq_BMS2_Orion_Error = TRUE THEN
	gq_BMS2_Error	:=	TRUE;
ELSE 
	gq_BMS2_Error	:=	FALSE;
END_IF
IF (gq_BMS1_Error = TRUE OR gq_BMS2_Error = TRUE) THEN
	gq_BMS_Error	:=	TRUE;
ELSE
	gq_BMS_Error	:=	FALSE;
END_IF
{endregion}
(**********************************************************)

{region "DCDC"}
IF (gq_BelDCDC_flt_InputUV OR
	gq_BelDCDC_flt_InputOV OR
	(*gq_BelDCDC_flt_OutputUV OR*)
	gq_BelDCDC_flt_OutputOV OR
	(*gq_BelDCDC_flt_OutputOC OR*) (*Need to reenable this when possible*)
	gq_BelDCDC_flt_OTP OR
	gq_BelDCDC_flt_I2CFault OR
	gq_BelDCDC_flt_CANFault OR
	gq_BelDCDC_flt_EEPROM_CRCFault OR
	gq_BelDCDC_flt_ShortCircuit OR
	gq_BelDCDC_flt_ThermistorFault OR
	gq_BelDCDC_flt_Overload OR
	gq_BelDCDC_flt_OutputOVLatch OR
	gq_BelDCDC_flt_ReversePolarity OR
	gq_BelDCDC_war_CoolantOTP OR
	gq_BelDCDC_war_CurrentLimiting OR
	(*gq_BelDCDC_sts_UnitEnabled OR
	gq_BelDCDC_sts_Wakeup OR
	gq_BelDCDC_sts_Fault OR
	gq_BelDCDC_sts_LatchedFault OR
	gq_BelDCDC_sts_RemoteShutdown OR
	gq_BelDCDC_sts_StartupInitDone OR
	gq_BelDCDC_sts_InputOK OR
	gq_BelDCDC_sts_HVILOK OR
	gq_BelDCDC_sts_ReversePolarity OR
	gq_BelDCDC_sts_Hiccup OR*)
	gq_BELDCDC_CommsLoss				) THEN
		gq_DCDC_Bel_Error	:=	TRUE;
ELSE
		gq_DCDC_Bel_Error	:=	FALSE;
END_IF
{endregion}
(**********************************************************)
{region "MCU"}
IF (gq_MCU_Fault_PhaseToChassis OR
	gq_MCU_Fault_InterlockBatteryCable OR
	gq_MCU_Fault_InterlockMotorCable OR
	gq_MCU_Fault_DriveCoverWasOpened OR
	gq_MCU_Fault_PhaseToChassisStatus OR
	(gq_MCU_CommsLoss = TRUE AND gu8_SystemState = DRIVE_SYS)) THEN
		gq_MCU_Error	:=	TRUE;
ELSE
		gq_MCU_Error	:=	FALSE;
END_IF
{endregion}
(**********************************************************)
{region "Charger"}
IF (gu8_ChargerType = CHARGER_BRUSA) THEN
	{region "NLG1"}
	IF (Brusa1_Rx.E_WrongHW OR
		Brusa1_Rx.E_WrongFPGA OR
		Brusa1_Rx.E_EPGAInit OR
		Brusa1_Rx.E_NVSRam OR
		Brusa1_Rx.E_Flash OR
		Brusa1_Rx.E_OSTrap OR
		Brusa1_Rx.E_HVIsoPos OR
		Brusa1_Rx.E_HVIsoNeg OR
		Brusa1_Rx.E_Internal OR
		Brusa1_Rx.E_TempInt OR
		Brusa1_Rx.E_DCHVVoltRed OR
		Brusa1_Rx.E_IntSupply OR
		Brusa1_Rx.E_CANMsgLost OR
		Brusa1_Rx.E_CANValue OR
		Brusa1_Rx.E_ACInterruption OR
		Brusa1_Rx.E_DCHVVoltRange OR
		Brusa1_Rx.E_TempCon OR
		Brusa1_Rx.E_ConLocked OR
		Brusa1_Rx.E_Interlock OR
		Brusa1_Rx.E_Crash OR
		Brusa1_Rx.E_PRELOAD OR
		Brusa1_Rx.E_BURST OR
		Brusa1_Rx.E_TPON OR
		Brusa1_Rx.E_UZK OR
		Brusa1_Rx.E_LatchFPGA OR
		Brusa1_Rx.E_OverTemp OR(*
		Brusa1_Rx.W_Watchdog OR
		(*Brusa1_Rx.W_PowRed OR*)
		Brusa1_Rx.W_TempInt OR
		Brusa1_Rx.W_CANTimeout OR
		Brusa1_Rx.W_CANOff OR
		Brusa1_Rx.W_CANRx OR
		Brusa1_Rx.W_CANTx OR
		Brusa1_Rx.W_ConLocked OR
		Brusa1_Rx.W_FPGA OR
		Brusa1_Rx.W_ACVoltage OR
		Brusa1_Rx.W_ACFrequency OR
		Brusa1_Rx.W_PRELOAD			*)
		Brusa1_Rx.CommsLoss = TRUE) THEN
			gq_NLG1_Error	:=	TRUE;
	ELSE
			gq_NLG1_Error	:=	FALSE;
	END_IF
	{endregion}
	{region "NLG2"}
	IF (Brusa2_Rx.E_WrongHW OR
		Brusa2_Rx.E_WrongFPGA OR
		Brusa2_Rx.E_EPGAInit OR
		Brusa2_Rx.E_NVSRam OR
		Brusa2_Rx.E_Flash OR
		Brusa2_Rx.E_OSTrap OR
		Brusa2_Rx.E_HVIsoPos OR
		Brusa2_Rx.E_HVIsoNeg OR
		Brusa2_Rx.E_Internal OR
		Brusa2_Rx.E_TempInt OR
		Brusa2_Rx.E_DCHVVoltRed OR
		Brusa2_Rx.E_IntSupply OR
		Brusa2_Rx.E_CANMsgLost OR
		Brusa2_Rx.E_CANValue OR
		Brusa2_Rx.E_ACInterruption OR
		Brusa2_Rx.E_DCHVVoltRange OR
		Brusa2_Rx.E_TempCon OR
		Brusa2_Rx.E_ConLocked OR
		Brusa2_Rx.E_Interlock OR
		Brusa2_Rx.E_Crash OR
		Brusa2_Rx.E_PRELOAD OR
		Brusa2_Rx.E_BURST OR
		Brusa2_Rx.E_TPON OR
	    Brusa2_Rx.E_UZK OR
		Brusa2_Rx.E_LatchFPGA OR
		Brusa2_Rx.E_OverTemp OR(*
		gq_NLG2_W_Watchdog OR
		(*gq_NLG2_W_PowRed OR*)
		gq_NLG2_W_TempInt OR
		gq_NLG2_W_CANTimeout OR
		gq_NLG2_W_CANOff OR
		gq_NLG2_W_CANRx OR
		gq_NLG2_W_CANTx OR
		gq_NLG2_W_ConLocked OR
		gq_NLG2_W_FPGA OR
		gq_NLG2_W_ACVoltage OR
		gq_NLG2_W_ACFrequency OR
		gq_NLG2_W_PRELOAD		*)
		Brusa2_Rx.CommsLoss = TRUE) THEN
			gq_NLG2_Error	:=	TRUE;
	ELSE
			gq_NLG2_Error	:=	FALSE;
	END_IF 
	{endregion}
END_IF
{endregion}
(**********************************************************)	 
{region "Sevcons"}
IF (gu8_Sevcon1_InverterStatus = FAULTOFF_STAT OR
	(gq_Sevcon1_CommsLoss = TRUE AND gu8_SystemState = DRIVE_SYS)) THEN
	gq_Sevcon_Steer_Error	:=	TRUE;
ELSE
	gq_Sevcon_Steer_Error	:=	FALSE;
END_IF
IF (gu8_Sevcon2_InverterStatus = FAULTOFF_STAT OR
	(gq_Sevcon2_CommsLoss = TRUE AND gu8_SystemState = DRIVE_SYS)) THEN
	gq_Sevcon_Compressor_Error	:=	TRUE;
ELSE
	gq_Sevcon_Compressor_Error	:=	FALSE;
END_IF
{endregion}
	 
{region "EPEC"}
IF ((SUPPLY_Power1/100) < 18 (*Change this back to 22*)) THEN (*SUPPLY_Power1*)
	gq_LV_Error	:=	TRUE;
ELSE
	gq_LV_Error	:=	FALSE; 
END_IF
{endregion}
 
 {region "Dennis"}
 IF ((gq_Dennis_CAN1_CommsLoss = TRUE OR CAN4_Rx.Handbrake_Rx_Timer.Q = TRUE) AND
	  gu8_ChassisType = CHASSIS_DENNIS AND gu8_SystemState = DRIVE_SYS) THEN
	hq_Dennis_CommsErr	:=	TRUE;
 ELSE
	hq_Dennis_CommsErr	:=	FALSE;	  
 END_IF
 {endregion}
	 
IF (gq_BMS_Error			OR
	gq_DCDC_Bel_Error		OR
	gq_MCU_Error			OR
	gq_NLG1_Error			OR
	gq_NLG2_Error 			OR
	gq_Sevcon_Steer_Error	OR
	gq_Sevcon_Compressor_Error OR
	gq_LV_Error OR
	hq_Dennis_CommsErr OR
	gq_EStop						) THEN
		gq_SystemError	:=	TRUE;
ELSE
		gq_SystemError	:=	FALSE;
END_IF


(*IF (gu16_BMS_LowCellVoltage < 26000) THEN
	hton_DriveMode_CutOff_Timer(IN := TRUE, PT := T#2S);
	hton_MCU_CutOff_Timer(IN := TRUE, PT := T#30S);
	(*hton_LowCVRecovery_Timer(IN := FALSE, PT := T#0S);*)
ELSIF (gu16_BMS_LowCellVoltage < 29000) THEN
	hton_MCU_CutOff_Timer(IN := TRUE, PT := T#30S);
	hton_DriveMode_CutOff_Timer(IN := FALSE, PT := T#0S); 
	+532
	(*hton_LowCVRecovery_Timer(IN := FALSE, PT := T#0S);*)
ELSE
	(*hton_LowCVRecovery_Timer(IN := TRUE, PT := T#5S);*)
	(*IF (hton_LowCVRecovery_Timer.Q = TRUE) THEN*)
		hton_MCU_CutOff_Timer(IN := FALSE, PT := T#0S);
		hton_DriveMode_CutOff_Timer(IN := FALSE, PT := T#0S);
	(*END_IF*)
END_IF

IF (hton_MCU_CutOff_Timer.Q = TRUE) THEN
	gq_MCU_CutOff_LowCellV	:=	TRUE;
END_IF

IF (hton_DriveMode_CutOff_Timer.Q = TRUE) THEN
	gq_DriveMode_CutOff_LowCellV	:=	TRUE;
END_IF*)

END_PROGRAM

// Application/UserCode/Main Program/System_StateSpace
PROGRAM System_StateSpace
VAR
	hton_Startup_Timer	:	TON;
	hq_StartupVoltage_Acceptable	:	BOOL;
END_VAR
VAR CONSTANT
	// IM
	PRECHARGE_START_VOLTAGE	:	USINT	:=	250;
	
	(*Charger plug in states*)
	CHARGER_DETECTED	:	USINT	:=	0;
	CHARGER_NOTCONNECTED		:	USINT	:=	5;
END_VAR

(*System state space with transitions*)


IF (gu8_SystemState = STANDBY_SYS) THEN
	hton_Startup_Timer(IN := TRUE, PT := T#5S);
	IF (hton_Startup_Timer.Q = TRUE AND DO_q_BatteryDischargeMain_DO = FALSE AND
		DO_q_Battery1ChargeMain_DO = FALSE AND DO_q_Battery2ChargeMain_DO = FALSE) THEN
		IF (DI_q_VehicleKL15_DI = TRUE AND hq_StartupVoltage_Acceptable = TRUE AND Brusa1_Rx.StatusPP = CHARGER_NOTCONNECTED AND
			gq_DriveMode_CutOff_LowCellV = FALSE) THEN
			gu8_SystemState := DRIVE_SYS;
		ELSIF (Brusa1_Rx.StatusPP = CHARGER_DETECTED) THEN
			gu8_SystemState := PLUGIN_SYS;
		ELSIF (gq_SystemError = TRUE OR gq_EStop = TRUE) THEN
			gu8_SystemState := ERROR_SYS;
		ELSE
			gu8_SystemState	:=	STANDBY_SYS;
		END_IF
	ELSE
		gu8_SystemState	:=	STANDBY_SYS;
	END_IF
	DO_q_ChargersWakeup_DO	:=	FALSE;
	gq_InitialProtocolGrab	:=	FALSE;
ELSIF (gu8_SystemState = DRIVE_SYS) THEN
	hton_Startup_Timer(IN	:=	FALSE, PT := T#0S);
	IF ((gq_SystemError = TRUE AND gq_HandBrake = TRUE) OR gq_EStop = TRUE) THEN
		gu8_SystemState := ERROR_SYS;
	ELSIF (Brusa1_Rx.StatusPP = CHARGER_DETECTED) THEN
		gu8_SystemState	:=	STANDBY_SYS;
	ELSIF (DI_q_VehicleKL15_DI = TRUE AND (Brusa1_Rx.StatusPP = CHARGER_NOTCONNECTED) AND gq_DriveMode_CutOff_LowCellV = FALSE) THEN
		gu8_SystemState := DRIVE_SYS;
	ELSE
		;IF (ABS(gr_VehicleSpeed_kmph) < 0.5) THEN
			gu8_SystemState	:=	STANDBY_SYS;
		END_IF
	END_IF
	DO_q_ChargersWakeup_DO	:=	FALSE;
ELSIF (gu8_SystemState = PLUGIN_SYS) THEN
	hton_Startup_Timer(IN	:=	FALSE, PT := T#0S);
	IF (gq_SystemError = TRUE OR gq_EStop = TRUE) THEN
		gu8_SystemState := ERROR_SYS;
	ELSIF (Brusa1_Rx.StatusPP = CHARGER_DETECTED) THEN
		gu8_SystemState	:=	PLUGIN_SYS; (*Stay in charge*)
	ELSIF ((Brusa1_Rx.StatusPP = CHARGER_NOTCONNECTED) AND DI_q_VehicleKL15_DI = TRUE AND hq_StartupVoltage_Acceptable = TRUE) THEN
		gu8_SystemState	:=	STANDBY_SYS; (*Go to drive*)
	ELSIF (Brusa1_Rx.StatusPP = CHARGER_NOTCONNECTED) THEN
		gu8_SystemState	:=	STANDBY_SYS; (*Go to standby*)
	
	END_IF
	DO_q_ChargersWakeup_DO	:=	TRUE;
	gq_InitialProtocolGrab	:=	FALSE;
ELSIF (gu8_SystemState = ERROR_SYS) THEN
	IF (gq_EStop = TRUE) THEN
		gq_EStopLatch	:=	TRUE; (*Stay in error until power is cycled*)
	END_IF
	(*There are no state transitions out of this state*)
	(*Only an overide will be able to transition out, tbd*)
	DO_q_ChargersWakeup_DO	:=	FALSE;
	gq_InitialProtocolGrab	:=	FALSE;
END_IF


(*Check to see if drive can be entered when the voltage across the HV components is low enough*)
IF (gr_Sevcon1_DCLink_Voltage < PRECHARGE_START_VOLTAGE AND
	gr_Sevcon2_DCLink_Voltage < PRECHARGE_START_VOLTAGE AND 
	gu16_MCU_HighPowerVoltage < PRECHARGE_START_VOLTAGE) THEN
	hq_StartupVoltage_Acceptable	:=	TRUE;
ELSE
	hq_StartupVoltage_Acceptable	:=	FALSE;
END_IF

END_PROGRAM

// Application/UserCode/Contactor Control/ContactorControl
PROGRAM ContactorControl
VAR
	hq_Test	:	BOOL;
	hton_Precharge_Timer	:	TON;
	hton_PrechargeDisconnect_Timer	:	TON;
	hton_PrechargeDisconnectBMS1_Timer	:	TON;
	hton_PrechargeDisconnectBMS2_Timer	:	TON;
	hton_MainContactorConnection_Delay	:	TON;
	
	hq_BatteryDischargeMain_Rq		:	BOOL	:=	FALSE;
	hq_Battery1ChargePrecharge_Rq	:	BOOL;
	hq_Battery1ChargeMain_Rq		:	BOOL;
	hq_Battery2ChargePrecharge_Rq	:	BOOL;
	hq_Battery2ChargeMain_Rq		:	BOOL;
	hq_BatteryDischargePrecharge_Rq	:	BOOL;
	
	hr_MainConnectionVoltage		:	REAL;
	
	hton_Contactor_Delay			:	TON;
	hq_TestPause	:	BOOL	:=	FALSE;
END_VAR
VAR CONSTANT
	CURRENT_DISCONNECT	:	SINT	:=	10; (*Only disconnect below 10Amps*)
	PRECHARGEEND_VOLTAGE_PERC	:	REAL	:=	0.95;
END_VAR


(*Non operational system state*)
IF (gu8_SystemState = STANDBY_SYS OR gu8_SystemState = ERROR_SYS OR gu8_SystemState = OFF_SYS (*OR hq_TestPause = FALSE This is a test trigger may be replaced later on with another on screen trigger*)) THEN
	hq_BatteryDischargeMain_Rq			:=	FALSE;
	hq_Battery1ChargePrecharge_Rq		:=	FALSE;
	hq_Battery1ChargeMain_Rq			:=	FALSE;
	hq_Battery2ChargePrecharge_Rq		:=	FALSE;
	hq_BatteryDischargePrecharge_Rq		:=	FALSE;
	hq_Battery2ChargeMain_Rq			:=	FALSE;
	hton_Precharge_Timer(IN := FALSE, PT := T#0MS);
	hton_PrechargeDisconnectBMS1_Timer(IN := FALSE, PT := T#0MS);
	hton_PrechargeDisconnectBMS2_Timer(IN := FALSE, PT := T#0MS);
	hton_Contactor_Delay(IN := FALSE, PT := T#0MS);
	
(*System State Discharge*)
ELSIF (gu8_SystemState = DRIVE_SYS AND gr_BMS_BatteryVoltage > 0) THEN
	hr_MainConnectionVoltage	:=	gr_BMS_BatteryVoltage * PRECHARGEEND_VOLTAGE_PERC;
	hton_Contactor_Delay(IN := TRUE, PT := T#500MS);
	IF (hton_Contactor_Delay.Q = TRUE) THEN
		IF ((gr_Sevcon1_DCLink_Voltage <= hr_MainConnectionVoltage OR gr_Sevcon2_DCLink_Voltage <= hr_MainConnectionVoltage OR
			gu16_MCU_HighPowerVoltage <= hr_MainConnectionVoltage) AND DO_q_BatteryDischargeMain_DO = FALSE) THEN
			hq_BatteryDischargePrecharge_Rq	:=	TRUE;
			hton_PrechargeDisconnect_Timer(IN := FALSE, PT := T#0MS);
			hton_MainContactorConnection_Delay(IN := FALSE, PT := T#0MS);
		ELSIF ((gr_Sevcon1_DCLink_Voltage > hr_MainConnectionVoltage AND gr_Sevcon2_DCLink_Voltage > hr_MainConnectionVoltage AND
				gu16_MCU_HighPowerVoltage > hr_MainConnectionVoltage) OR DO_q_BatteryDischargeMain_DO = TRUE) THEN
			hton_MainContactorConnection_Delay(IN := TRUE, PT := T#100MS);
			IF (hton_MainContactorConnection_Delay.Q = TRUE) THEN
				hq_BatteryDischargeMain_Rq		:=	TRUE;
				hton_PrechargeDisconnect_Timer(IN := TRUE, PT := T#1S);
				IF (hton_PrechargeDisconnect_Timer.Q = TRUE) THEN
					hq_BatteryDischargePrecharge_Rq	:=	FALSE;
				END_IF
			END_IF
		ELSE
			hq_BatteryDischargeMain_Rq		:=	FALSE;
		END_IF
	END_IF
	hq_Battery1ChargePrecharge_Rq		:=	FALSE;
	hq_Battery1ChargeMain_Rq			:=	FALSE;
	hq_Battery2ChargePrecharge_Rq		:=	FALSE;
	hq_Battery2ChargeMain_Rq			:=	FALSE;
	
(*System State Charge*)
ELSIF (gu8_SystemState = PLUGIN_SYS AND Brusa1_Rx.S_ACDet = TRUE AND Brusa2_Rx.S_ACDet = TRUE AND gr_BMS_BatteryVoltage > 0) THEN
	hton_Contactor_Delay(IN := DO_q_DrivetrainKL15C_DO, PT := T#500MS);
	IF (hton_Contactor_Delay.Q = TRUE) THEN
	
	    // Check that BMS1 safety is ok
		IF OrionBMS1_RxConversion.Safety_OK THEN
			IF (Brusa1_RxConversion.DCHVVoltAct <= (gr_BMS1_Voltage * PRECHARGEEND_VOLTAGE_PERC) AND (DO_q_Battery1ChargeMain_DO = FALSE)) THEN
				hq_Battery1ChargePrecharge_Rq		  := TRUE;
			ELSIF (Brusa1_RxConversion.DCHVVoltAct > (gr_BMS1_Voltage * PRECHARGEEND_VOLTAGE_PERC) OR DO_q_Battery1ChargeMain_DO) THEN
				hq_Battery1ChargeMain_Rq			  := TRUE;
				hton_PrechargeDisconnectBMS1_Timer(IN := TRUE, PT := T#1S);
				IF (hton_PrechargeDisconnectBMS1_Timer.Q) THEN
						hq_Battery1ChargePrecharge_Rq := FALSE;
				END_IF
			END_IF
		END_IF
		
		// Check that BMS2 safety is ok
		IF OrionBMS2_RxConversion.Safety_OK THEN
			IF (Brusa1_RxConversion.DCHVVoltAct <= (gr_BMS2_Voltage * PRECHARGEEND_VOLTAGE_PERC) AND (DO_q_Battery2ChargeMain_DO = FALSE)) THEN
				hq_Battery2ChargePrecharge_Rq		  := TRUE;
			ELSIF (Brusa1_RxConversion.DCHVVoltAct > (gr_BMS2_Voltage * PRECHARGEEND_VOLTAGE_PERC) OR DO_q_Battery2ChargeMain_DO) THEN
				hq_Battery2ChargeMain_Rq			  := TRUE;	
				hton_PrechargeDisconnectBMS2_Timer(IN := TRUE, PT := T#1S);
				IF (hton_PrechargeDisconnectBMS2_Timer.Q) THEN
					hq_Battery2ChargePrecharge_Rq	  := FALSE;
				END_IF
			END_IF
		END_IF
		
	ELSE
		hq_Battery1ChargePrecharge_Rq		:=	FALSE;
		hq_Battery2ChargePrecharge_Rq		:=	FALSE;
		hq_Battery1ChargeMain_Rq			:=	FALSE;
		hq_Battery2ChargeMain_Rq			:=	FALSE;
	END_IF
	(*Ensure discharge contactors are open*)
	hq_BatteryDischargeMain_Rq		:=	FALSE;
	hq_BatteryDischargePrecharge_Rq	:=	FALSE;
ELSE
	hq_BatteryDischargeMain_Rq			:=	FALSE;
	hq_Battery1ChargePrecharge_Rq		:=	FALSE;
	hq_Battery1ChargeMain_Rq			:=	FALSE;
	hq_Battery2ChargePrecharge_Rq		:=	FALSE;
	hq_BatteryDischargePrecharge_Rq		:=	FALSE;
	hq_Battery2ChargeMain_Rq			:=	FALSE;
	hton_Precharge_Timer(IN := FALSE, PT := T#0MS);
	hton_Contactor_Delay(IN := FALSE, PT := T#0MS);
END_IF


(*Set the actual output values*)
(*Current protection so if system current is over a certain value maintain contactor state to prevent welds*)
IF ((DOS_q_BatteryDischargeMain_DO <> hq_BatteryDischargeMain_Rq) AND (ABS(gs16_BMS_BatteryCurrent) > CONTACTORSWITCH_CURRENT_LIMIT)) THEN
	DO_q_BatteryDischargeMain_DO	:=	DOS_q_BatteryDischargeMain_DO;
ELSE
	DO_q_BatteryDischargeMain_DO	:=	hq_BatteryDischargeMain_Rq;
END_IF

IF ((DOS_q_Battery1ChargeMain_DO <> hq_Battery1ChargeMain_Rq) AND (ABS(gs16_BMS_BatteryCurrent) > CONTACTORSWITCH_CURRENT_LIMIT)) THEN
	DO_q_Battery1ChargeMain_DO	:=	FALSE(*DOS_q_Battery1ChargeMain_DO*); (*FALSE if cable doesnt sort*)
ELSE
	DO_q_Battery1ChargeMain_DO	:=	hq_Battery1ChargeMain_Rq;
END_IF

IF (DOS_q_Battery1ChargeMain_DO <> hq_Battery2ChargeMain_Rq AND (ABS(gs16_BMS_BatteryCurrent) > CONTACTORSWITCH_CURRENT_LIMIT)) THEN
	DO_q_Battery2ChargeMain_DO	:=	DOS_q_Battery2ChargeMain_DO;
ELSE
	DO_q_Battery2ChargeMain_DO	:=	hq_Battery2ChargeMain_Rq;
END_IF
(*Precharge contactors can change states to allow system connection*)
DO_q_BatteryDischargePrecharge_DO	:=	hq_BatteryDischargePrecharge_Rq;
DO_q_Battery1ChargePrecharge_DO		:=	hq_Battery1ChargePrecharge_Rq;
DO_q_Battery2ChargePrecharge_DO		:=	hq_Battery2ChargePrecharge_Rq;


(*
DO_q_ChargePlugLockPulse_DO
DO_q_ChargePlugLockPosition_DO
DI_q_ChargePlugLockStatus_DI
*)

END_PROGRAM

// Application/UserCode/MCU/GearSelection
PROGRAM GearSelection
VAR
END_VAR

(*Do I need to ensure low speed for gear change*)
(*ADDED minimal vehicle speed to gear selection*)

